    !Tr_meulage_bavure : Meulage de la bavure
    LOCAL CONST Robtarget Tr_meulage_bavure_0 := [[-72.96559375,77.9778671875,80.7656328125],[0.524498637144303,-0.433871580767109,0.466936666004684,-0.564470354382628],[0,0,0,0],[8.999999E+09,8.999999E+09,8.999999E+09,8.999999E+09,8.999999E+09,8.999999E+09]];
    LOCAL CONST Robtarget Tr_meulage_bavure_1 := [[-73.4128125,91.0669140625,78.9180078125],[0.519154027655531,-0.429298696043106,0.470963403699329,-0.569539460898604],[0,0,0,0],[8.999999E+09,8.999999E+09,8.999999E+09,8.999999E+09,8.999999E+09,8.999999E+09]];
    LOCAL CONST Robtarget Tr_meulage_bavure_2 := [[-73.421484375,92.5101640625,78.714984375],[0.502366205049294,-0.414981939275173,0.483103622109588,-0.584832519961385],[0,0,0,0],[8.999999E+09,8.999999E+09,8.999999E+09,8.999999E+09,8.999999E+09,8.999999E+09]];
    LOCAL CONST Robtarget Tr_meulage_bavure_3 := [[-73.3546796875,94.05434375,78.4991015625],[0.471901589556323,-0.389165581198061,0.503332600241078,-0.610340342529925],[0,0,0,0],[8.999999E+09,8.999999E+09,8.999999E+09,8.999999E+09,8.999999E+09,8.999999E+09]];
    LOCAL CONST Robtarget Tr_meulage_bavure_4 := [[-73.06753125,95.5965546875,78.2873359375],[0.424855473704573,-0.349592797660536,0.530576857987408,-0.644802993212153],[0,0,0,0],[8.999999E+09,8.999999E+09,8.999999E+09,8.999999E+09,8.999999E+09,8.999999E+09]];
    LOCAL CONST Robtarget Tr_meulage_bavure_5 := [[-72.49625,97.5792109375,78.0186171875],[0.360143668564367,-0.295563225119298,0.561336594654554,-0.683988410319727],[0,0,0,0],[8.999999E+09,8.999999E+09,8.999999E+09,8.999999E+09,8.999999E+09,8.999999E+09]];
    LOCAL CONST Robtarget Tr_meulage_bavure_6 := [[-71.18978125,99.7963125,77.72978125],[0.282652351555885,-0.231289577368078,0.589537581877902,-0.720456951603897],[0,0,0,0],[8.999999E+09,8.999999E+09,8.999999E+09,8.999999E+09,8.999999E+09,8.999999E+09]];
    LOCAL CONST Robtarget Tr_meulage_bavure_7 := [[-69.0200625,100.7901796875,77.627953125],[0.204414557432899,-0.166757138111491,0.609729609191989,-0.747419928335445],[0,0,0,0],[8.999999E+09,8.999999E+09,8.999999E+09,8.999999E+09,8.999999E+09,8.999999E+09]];
    LOCAL CONST Robtarget Tr_meulage_bavure_8 := [[-65.746828125,102.36953125,77.46309375],[0.137940363092354,-0.112187700081668,0.620915411831161,-0.763446414315291],[0,0,0,0],[8.999999E+09,8.999999E+09,8.999999E+09,8.999999E+09,8.999999E+09,8.999999E+09]];
    LOCAL CONST Robtarget Tr_meulage_bavure_9 := [[-61.93778515625,102.33946875,77.5338046875],[0.0895913508579802,-0.0726567540841667,0.625676522996422,-0.771507144820126],[0,0,0,0],[8.999999E+09,8.999999E+09,8.999999E+09,8.999999E+09,8.999999E+09,8.999999E+09]];
    LOCAL CONST Robtarget Tr_meulage_bavure_10 := [[-57.10214453125,102.293921875,77.6246171875],[0.0599889984484553,-0.0485258607399388,0.627036256816005,-0.775159398796642],[0,0,0,0],[8.999999E+09,8.999999E+09,8.999999E+09,8.999999E+09,8.999999E+09,8.999999E+09]];
    LOCAL CONST Robtarget Tr_meulage_bavure_11 := [[-55.68121484375,102.1337578125,77.6719296875],[0.047095653965774,-0.0380159924114396,0.626957544520652,-0.776698796875046],[0,0,0,0],[8.999999E+09,8.999999E+09,8.999999E+09,8.999999E+09,8.999999E+09,8.999999E+09]];
    LOCAL CONST Robtarget Tr_meulage_bavure_12 := [[-51.0949140625,101.74665625,77.8063984375],[0.0480334258632763,-0.0387120379923225,0.626315605146604,-0.777124784615805],[0,0,0,0],[8.999999E+09,8.999999E+09,8.999999E+09,8.999999E+09,8.999999E+09,8.999999E+09]];
    LOCAL CONST Robtarget Tr_meulage_bavure_13 := [[-49.12283984375,101.942609375,77.8132734375],[0.0593251793460015,-0.0477669656022839,0.625326539875387,-0.77663734047507],[0,0,0,0],[8.999999E+09,8.999999E+09,8.999999E+09,8.999999E+09,8.999999E+09,8.999999E+09]];
    LOCAL CONST Robtarget Tr_meulage_bavure_14 := [[-44.2636640625,102.2745859375,77.8514296875],[0.0768851540962994,-0.0618884366060826,0.62398012963373,-0.7751821026806],[0,0,0,0],[8.999999E+09,8.999999E+09,8.999999E+09,8.999999E+09,8.999999E+09,8.999999E+09]];
    LOCAL CONST Robtarget Tr_meulage_bavure_15 := [[-42.5008984375,102.301234375,77.878453125],[0.0961771542647169,-0.0774482725613951,0.622392974176696,-0.772902778989882],[0,0,0,0],[8.999999E+09,8.999999E+09,8.999999E+09,8.999999E+09,8.999999E+09,8.999999E+09]];
    LOCAL CONST Robtarget Tr_meulage_bavure_16 := [[-41.74234765625,102.4241171875,77.874421875],[0.112993286570119,-0.0910887399273819,0.620961489830233,-0.770287080766867],[0,0,0,0],[8.999999E+09,8.999999E+09,8.999999E+09,8.999999E+09,8.999999E+09,8.999999E+09]];
    LOCAL CONST Robtarget Tr_meulage_bavure_17 := [[-41.52457421875,102.525171875,77.864015625],[0.12430618580482,-0.100382813703911,0.620196366080517,-0.768002428631619],[0,0,0,0],[8.999999E+09,8.999999E+09,8.999999E+09,8.999999E+09,8.999999E+09,8.999999E+09]];
    LOCAL CONST Robtarget Tr_meulage_bavure_18 := [[-38.44026171875,103.5358046875,77.775796875],[0.128536780570744,-0.104042680848259,0.620496098458886,-0.766575507304868],[0,0,0,0],[8.999999E+09,8.999999E+09,8.999999E+09,8.999999E+09,8.999999E+09,8.999999E+09]];
    LOCAL CONST Robtarget Tr_meulage_bavure_19 := [[-35.635421875,105.1262265625,77.601203125],[0.125456426611608,-0.101841270384386,0.621966700070119,-0.766189574891376],[0,0,0,0],[8.999999E+09,8.999999E+09,8.999999E+09,8.999999E+09,8.999999E+09,8.999999E+09]];
    LOCAL CONST Robtarget Tr_meulage_bavure_20 := [[-32.589919921875,106.671859375,77.4371015625],[0.115819970243643,-0.0943317978781946,0.624426753397045,-0.766667122057451],[0,0,0,0],[8.999999E+09,8.999999E+09,8.999999E+09,8.999999E+09,8.999999E+09,8.999999E+09]];
    LOCAL CONST Robtarget Tr_meulage_bavure_21 := [[-30.991841796875,107.5399765625,77.3429765625],[0.1010430938105,-0.0826008420732401,0.627499640971008,-0.767601195063719],[0,0,0,0],[8.999999E+09,8.999999E+09,8.999999E+09,8.999999E+09,8.999999E+09,8.999999E+09]];
    LOCAL CONST Robtarget Tr_meulage_bavure_22 := [[-30.700533203125,107.67775,77.3286953125],[0.0830195632788944,-0.0681360313903383,0.630743998534626,-0.768522765864427],[0,0,0,0],[8.999999E+09,8.999999E+09,8.999999E+09,8.999999E+09,8.999999E+09,8.999999E+09]];
    LOCAL CONST Robtarget Tr_meulage_bavure_23 := [[-26.497271484375,109.0772421875,77.20534375],[0.0639091173605292,-0.0526684914647995,0.633792076669562,-0.769057382953902],[0,0,0,0],[8.999999E+09,8.999999E+09,8.999999E+09,8.999999E+09,8.999999E+09,8.999999E+09]];
    LOCAL CONST Robtarget Tr_meulage_bavure_24 := [[-26.031384765625,109.2446875,77.1899453125],[0.0458469341804628,-0.0379425139443275,0.63643994137898,-0.769027064074703],[0,0,0,0],[8.999999E+09,8.999999E+09,8.999999E+09,8.999999E+09,8.999999E+09,8.999999E+09]];
    LOCAL CONST Robtarget Tr_meulage_bavure_25 := [[-24.007275390625,109.3088125,77.2162578125],[0.0305658967448666,-0.0254025527691808,0.638653823464502,-0.768467130099371],[0,0,0,0],[8.999999E+09,8.999999E+09,8.999999E+09,8.999999E+09,8.999999E+09,8.999999E+09]];
    LOCAL CONST Robtarget Tr_meulage_bavure_26 := [[-22.2173125,109.3889609375,77.236234375],[0.0190622543195306,-0.015907517289484,0.640516947745874,-0.767542585791988],[0,0,0,0],[8.999999E+09,8.999999E+09,8.999999E+09,8.999999E+09,8.999999E+09,8.999999E+09]];
    LOCAL CONST Robtarget Tr_meulage_bavure_27 := [[-19.49805859375,109.3278828125,77.2922890625],[0.0115387164285388,-0.00966712028603791,0.642129419226901,-0.76644844169186],[0,0,0,0],[8.999999E+09,8.999999E+09,8.999999E+09,8.999999E+09,8.999999E+09,8.999999E+09]];
    LOCAL CONST Robtarget Tr_meulage_bavure_28 := [[-15.033275390625,109.3440546875,77.3679453125],[0.00752164158955457,-0.00632501640817029,0.643568832555467,-0.765325144522528],[0,0,0,0],[8.999999E+09,8.999999E+09,8.999999E+09,8.999999E+09,8.999999E+09,8.999999E+09]];
    LOCAL CONST Robtarget Tr_meulage_bavure_29 := [[-11.9529951171875,109.418640625,77.4112265625],[0.006151571426882,-0.00519059536474067,0.644865070540276,-0.764254052449723],[0,0,0,0],[8.999999E+09,8.999999E+09,8.999999E+09,8.999999E+09,8.999999E+09,8.999999E+09]];
    LOCAL CONST Robtarget Tr_meulage_bavure_30 := [[-3.52283715820313,109.6361953125,77.527796875],[0.00643709893464829,-0.00544820591259924,0.646018072081297,-0.763275527810242],[0,0,0,0],[8.999999E+09,8.999999E+09,8.999999E+09,8.999999E+09,8.999999E+09,8.999999E+09]];
    LOCAL CONST Robtarget Tr_meulage_bavure_31 := [[2.07959692382813,109.6801015625,77.619421875],[0.00754756157762624,-0.0064053255495668,0.647024086186714,-0.762405297734141],[0,0,0,0],[8.999999E+09,8.999999E+09,8.999999E+09,8.999999E+09,8.999999E+09,8.999999E+09]];
    LOCAL CONST Robtarget Tr_meulage_bavure_32 := [[10.4173935546875,109.9232578125,77.7307734375],[0.0089059924357084,-0.00757553932592323,0.64787449029423,-0.761657363470378],[0,0,0,0],[8.999999E+09,8.999999E+09,8.999999E+09,8.999999E+09,8.999999E+09,8.999999E+09]];
    LOCAL CONST Robtarget Tr_meulage_bavure_33 := [[14.9681103515625,110.080015625,77.788171875],[0.0101637625195787,-0.00866164743259205,0.648566021431958,-0.761041253572446],[0,0,0,0],[8.999999E+09,8.999999E+09,8.999999E+09,8.999999E+09,8.999999E+09,8.999999E+09]];
    LOCAL CONST Robtarget Tr_meulage_bavure_34 := [[17.49816015625,110.1214765625,77.8265078125],[0.011196506180603,-0.00955583886393558,0.649107385814113,-0.760554354319612],[0,0,0,0],[8.999999E+09,8.999999E+09,8.999999E+09,8.999999E+09,8.999999E+09,8.999999E+09]];
    LOCAL CONST Robtarget Tr_meulage_bavure_35 := [[19.417255859375,110.1771171875,77.8521875],[0.0119919328824449,-0.0102458555270846,0.649505699878697,-0.760193108239838],[0,0,0,0],[8.999999E+09,8.999999E+09,8.999999E+09,8.999999E+09,8.999999E+09,8.999999E+09]];
    LOCAL CONST Robtarget Tr_meulage_bavure_36 := [[28.539337890625,110.462484375,77.9713046875],[0.0126142416671802,-0.0107855693015085,0.64977613721374,-0.759944421592524],[0,0,0,0],[8.999999E+09,8.999999E+09,8.999999E+09,8.999999E+09,8.999999E+09,8.999999E+09]];
    LOCAL CONST Robtarget Tr_meulage_bavure_37 := [[30.24216796875,110.5603125,77.9872734375],[0.0132183794150829,-0.0113071132675388,0.64993291030976,-0.759792495179756],[0,0,0,0],[8.999999E+09,8.999999E+09,8.999999E+09,8.999999E+09,8.999999E+09,8.999999E+09]];
    LOCAL CONST Robtarget Tr_meulage_bavure_38 := [[35.8308828125,110.707703125,78.064109375],[0.0140329277622215,-0.0120062947243841,0.649995732976522,-0.759713415004451],[0,0,0,0],[8.999999E+09,8.999999E+09,8.999999E+09,8.999999E+09,8.999999E+09,8.999999E+09]];
    LOCAL CONST Robtarget Tr_meulage_bavure_39 := [[41.86768359375,110.7581015625,78.1623984375],[0.0153254201090454,-0.0131126639284937,0.649989769318002,-0.759675252542236],[0,0,0,0],[8.999999E+09,8.999999E+09,8.999999E+09,8.999999E+09,8.999999E+09,8.999999E+09]];
    LOCAL CONST Robtarget Tr_meulage_bavure_40 := [[48.0332890625,110.8994453125,78.2501484375],[0.0173576592937217,-0.0148509775353596,0.649939701863269,-0.759642379065289],[0,0,0,0],[8.999999E+09,8.999999E+09,8.999999E+09,8.999999E+09,8.999999E+09,8.999999E+09]];
    LOCAL CONST Robtarget Tr_meulage_bavure_41 := [[54.3366640625,111.20328125,78.31746875],[0.0203296694220353,-0.0173934789408263,0.649869936126184,-0.759574379209091],[0,0,0,0],[8.999999E+09,8.999999E+09,8.999999E+09,8.999999E+09,8.999999E+09,8.999999E+09]];
    LOCAL CONST Robtarget Tr_meulage_bavure_42 := [[62.10978125,111.67840625,78.386359375],[0.0243160425327989,-0.0208061051968355,0.649805737683987,-0.75942632251921],[0,0,0,0],[8.999999E+09,8.999999E+09,8.999999E+09,8.999999E+09,8.999999E+09,8.999999E+09]];
    LOCAL CONST Robtarget Tr_meulage_bavure_43 := [[64.7070625,111.7126171875,78.426890625],[0.0292129223072121,-0.0250039510309742,0.649775145993782,-0.759153256761685],[0,0,0,0],[8.999999E+09,8.999999E+09,8.999999E+09,8.999999E+09,8.999999E+09,8.999999E+09]];
    LOCAL CONST Robtarget Tr_meulage_bavure_44 := [[71.0410703125,111.980734375,78.499765625],[0.0346206886603777,-0.0296511906304267,0.649815638883284,-0.758723830041992],[0,0,0,0],[8.999999E+09,8.999999E+09,8.999999E+09,8.999999E+09,8.999999E+09,8.999999E+09]];
    LOCAL CONST Robtarget Tr_meulage_bavure_45 := [[73.262921875,112.0517265625,78.5285703125],[0.0397101679776423,-0.034045022612306,0.649985629173882,-0.758144261247124],[0,0,0,0],[8.999999E+09,8.999999E+09,8.999999E+09,8.999999E+09,8.999999E+09,8.999999E+09]];
    LOCAL CONST Robtarget Tr_meulage_bavure_46 := [[76.461375,112.383578125,78.53775],[0.0431961175728289,-0.037089230175035,0.6503823304321,-0.757470335190342],[0,0,0,0],[8.999999E+09,8.999999E+09,8.999999E+09,8.999999E+09,8.999999E+09,8.999999E+09]];
    LOCAL CONST Robtarget Tr_meulage_bavure_47 := [[79.9172578125,112.976390625,78.51475],[0.0432055408652098,-0.0371729766684629,0.651142540142572,-0.756812290770195],[0,0,0,0],[8.999999E+09,8.999999E+09,8.999999E+09,8.999999E+09,8.999999E+09,8.999999E+09]];
    LOCAL CONST Robtarget Tr_meulage_bavure_48 := [[80.2113828125,113.0060625,78.5157109375],[0.037391914390404,-0.0322554155127835,0.652386719553825,-0.756275744063048],[0,0,0,0],[8.999999E+09,8.999999E+09,8.999999E+09,8.999999E+09,8.999999E+09,8.999999E+09]];
    LOCAL CONST Robtarget Tr_meulage_bavure_49 := [[80.3745,113.014796875,78.517328125],[0.0230149202058911,-0.0199173517811249,0.654084723143131,-0.755808697685278],[0,0,0,0],[8.999999E+09,8.999999E+09,8.999999E+09,8.999999E+09,8.999999E+09,8.999999E+09]];
    LOCAL CONST Robtarget Tr_meulage_bavure_50 := [[80.4332421875,113.017515625,78.51796875],[0.00296501442514855,-0.00257573271942405,-0.655805220899747,0.754919920608174],[0,0,0,0],[8.999999E+09,8.999999E+09,8.999999E+09,8.999999E+09,8.999999E+09,8.999999E+09]];
    LOCAL CONST Robtarget Tr_meulage_bavure_51 := [[80.6750703125,113.011046875,78.5231015625],[0.0435007280531674,-0.0379546708906836,-0.656343344232936,0.752250320104651],[0,0,0,0],[8.999999E+09,8.999999E+09,8.999999E+09,8.999999E+09,8.999999E+09,8.999999E+09]];
    LOCAL CONST Robtarget Tr_meulage_bavure_52 := [[84.2401953125,113.0950625,78.5735234375],[0.100430419351731,-0.0880538690704243,-0.653348955544318,0.745181447232627],[0,0,0,0],[8.999999E+09,8.999999E+09,8.999999E+09,8.999999E+09,8.999999E+09,8.999999E+09]];
    LOCAL CONST Robtarget Tr_meulage_bavure_53 := [[87.07825,112.6916484375,78.679765625],[0.171895999689374,-0.151514363982637,-0.64363944210562,0.730221494728616],[0,0,0,0],[8.999999E+09,8.999999E+09,8.999999E+09,8.999999E+09,8.999999E+09,8.999999E+09]];
    LOCAL CONST Robtarget Tr_meulage_bavure_54 := [[87.4928984375,112.534953125,78.70903125],[0.249895133589002,-0.221511120301779,-0.625251119447997,0.70536960766694],[0,0,0,0],[8.999999E+09,8.999999E+09,8.999999E+09,8.999999E+09,8.999999E+09,8.999999E+09]];
    LOCAL CONST Robtarget Tr_meulage_bavure_55 := [[90.6231484375,111.0967890625,78.9658203125],[0.322554687399856,-0.287599923412569,-0.600154409759069,0.673096903971641],[0,0,0,0],[8.999999E+09,8.999999E+09,8.999999E+09,8.999999E+09,8.999999E+09,8.999999E+09]];
    LOCAL CONST Robtarget Tr_meulage_bavure_56 := [[91.76803125,109.5467734375,79.2036796875],[0.381349520380913,-0.342059463322267,-0.573448074256001,0.639316176073321],[0,0,0,0],[8.999999E+09,8.999999E+09,8.999999E+09,8.999999E+09,8.999999E+09,8.999999E+09]];
    LOCAL CONST Robtarget Tr_meulage_bavure_57 := [[92.15846875,108.9862109375,79.2892890625],[0.424645892808707,-0.383169856962373,-0.549520170935442,0.609002716062263],[0,0,0,0],[8.999999E+09,8.999999E+09,8.999999E+09,8.999999E+09,8.999999E+09,8.999999E+09]];
    LOCAL CONST Robtarget Tr_meulage_bavure_58 := [[92.243578125,108.7665078125,79.32165625],[0.455045695708042,-0.412995099011091,-0.530193694826248,0.584177292418059],[0,0,0,0],[8.999999E+09,8.999999E+09,8.999999E+09,8.999999E+09,8.999999E+09,8.999999E+09]];
    LOCAL CONST Robtarget Tr_meulage_bavure_59 := [[92.5548515625,106.992625,79.5764296875],[0.475960918078303,-0.43438038951089,-0.515492981292442,0.564837912952607],[0,0,0,0],[8.999999E+09,8.999999E+09,8.999999E+09,8.999999E+09,8.999999E+09,8.999999E+09]];
    LOCAL CONST Robtarget Tr_meulage_bavure_60 := [[93.0728125,104.701171875,79.9075625],[0.490145484495864,-0.449643756910361,-0.504780923350693,0.550249139318793],[0,0,0,0],[8.999999E+09,8.999999E+09,8.999999E+09,8.999999E+09,8.999999E+09,8.999999E+09]];
    LOCAL CONST Robtarget Tr_meulage_bavure_61 := [[93.1247578125,104.1366484375,79.9878203125],[0.499440463656121,-0.460329556127368,-0.497407243630099,0.539668376878659],[0,0,0,0],[8.999999E+09,8.999999E+09,8.999999E+09,8.999999E+09,8.999999E+09,8.999999E+09]];
    LOCAL CONST Robtarget Tr_meulage_bavure_62 := [[93.0234140625,101.6530390625,80.3351484375],[0.50508155139008,-0.467466020070269,-0.492804195180393,0.532458610351694],[0,0,0,0],[8.999999E+09,8.999999E+09,8.999999E+09,8.999999E+09,8.999999E+09,8.999999E+09]];
    LOCAL CONST Robtarget Tr_meulage_bavure_63 := [[93.0410859375,95.376796875,81.2176640625],[0.50800153503494,-0.471840804312682,-0.49042003163118,0.528004629110937],[0,0,0,0],[8.999999E+09,8.999999E+09,8.999999E+09,8.999999E+09,8.999999E+09,8.999999E+09]];
    LOCAL CONST Robtarget Tr_meulage_bavure_64 := [[93.069375,92.16809375,81.6691796875],[0.509036100077303,-0.474181488278619,-0.489639528685966,0.525630380533839],[0,0,0,0],[8.999999E+09,8.999999E+09,8.999999E+09,8.999999E+09,8.999999E+09,8.999999E+09]];
    LOCAL CONST Robtarget Tr_meulage_bavure_65 := [[93.288359375,82.485171875,83.0340546875],[0.509017334222879,-0.475239181311407,-0.489764889439004,0.524575473197039],[0,0,0,0],[8.999999E+09,8.999999E+09,8.999999E+09,8.999999E+09,8.999999E+09,8.999999E+09]];
    LOCAL CONST Robtarget Tr_meulage_bavure_66 := [[93.3151640625,82.0066953125,83.1017734375],[0.50860623912965,-0.475631289271055,-0.49021362642387,0.524199552320589],[0,0,0,0],[8.999999E+09,8.999999E+09,8.999999E+09,8.999999E+09,8.999999E+09,8.999999E+09]];
    LOCAL CONST Robtarget Tr_meulage_bavure_67 := [[93.3164765625,78.2097265625,83.6355078125],[0.508254924988694,-0.475792756551136,-0.490579965834165,0.524051029156855],[0,0,0,0],[8.999999E+09,8.999999E+09,8.999999E+09,8.999999E+09,8.999999E+09,8.999999E+09]];
    LOCAL CONST Robtarget Tr_meulage_bavure_68 := [[93.3254765625,77.7136796875,83.705390625],[0.508152417130769,-0.475929318394814,-0.490695448122873,0.523918297111197],[0,0,0,0],[8.999999E+09,8.999999E+09,8.999999E+09,8.999999E+09,8.999999E+09,8.999999E+09]];
    LOCAL CONST Robtarget Tr_meulage_bavure_69 := [[93.335359375,76.9299453125,83.8157265625],[0.508272125765174,-0.47604503540112,-0.490587023385963,0.523798570946311],[0,0,0,0],[8.999999E+09,8.999999E+09,8.999999E+09,8.999999E+09,8.999999E+09,8.999999E+09]];
    LOCAL CONST Robtarget Tr_meulage_bavure_70 := [[93.519703125,69.4331171875,84.87271875],[0.508492654218718,-0.476062116804073,-0.490368503184077,0.523773627280561],[0,0,0,0],[8.999999E+09,8.999999E+09,8.999999E+09,8.999999E+09,8.999999E+09,8.999999E+09]];
    LOCAL CONST Robtarget Tr_meulage_bavure_71 := [[93.6854296875,57.159515625,86.6008125],[0.508666271307918,-0.47588743567968,-0.490178457605301,0.523941650086731],[0,0,0,0],[8.999999E+09,8.999999E+09,8.999999E+09,8.999999E+09,8.999999E+09,8.999999E+09]];
    LOCAL CONST Robtarget Tr_meulage_bavure_72 := [[93.70446875,56.32636328125,86.7182578125],[0.508704393662726,-0.475482573374445,-0.490101155326875,0.524344371413212],[0,0,0,0],[8.999999E+09,8.999999E+09,8.999999E+09,8.999999E+09,8.999999E+09,8.999999E+09]];
    LOCAL CONST Robtarget Tr_meulage_bavure_73 := [[93.7035234375,55.86555859375,86.783015625],[0.508602047574567,-0.4748831497868,-0.490143997412789,0.524946485893312],[0,0,0,0],[8.999999E+09,8.999999E+09,8.999999E+09,8.999999E+09,8.999999E+09,8.999999E+09]];
    LOCAL CONST Robtarget Tr_meulage_bavure_74 := [[93.8570078125,51.93498046875,87.3381796875],[0.508420795232722,-0.474188979834551,-0.490254414881032,0.525645997861728],[0,0,0,0],[8.999999E+09,8.999999E+09,8.999999E+09,8.999999E+09,8.999999E+09,8.999999E+09]];
    LOCAL CONST Robtarget Tr_meulage_bavure_75 := [[94.0242734375,48.27883203125,87.855015625],[0.508263944010555,-0.473534553785341,-0.490342733317366,0.526304848422478],[0,0,0,0],[8.999999E+09,8.999999E+09,8.999999E+09,8.999999E+09,8.999999E+09,8.999999E+09]];
    LOCAL CONST Robtarget Tr_meulage_bavure_76 := [[94.0660078125,47.71273828125,87.9353203125],[0.50823520319336,-0.473057952864069,-0.49032064057548,0.526781568482337],[0,0,0,0],[8.999999E+09,8.999999E+09,8.999999E+09,8.999999E+09,8.999999E+09,8.999999E+09]];
    LOCAL CONST Robtarget Tr_meulage_bavure_77 := [[94.2361953125,44.8235,88.34440625],[0.508411095050095,-0.472850003528543,-0.490122652940176,0.526982748928183],[0,0,0,0],[8.999999E+09,8.999999E+09,8.999999E+09,8.999999E+09,8.999999E+09,8.999999E+09]];
    LOCAL CONST Robtarget Tr_meulage_bavure_78 := [[94.49140625,41.3637890625,88.8351640625],[0.508810216422261,-0.472937041493102,-0.489733748977065,0.526880986144834],[0,0,0,0],[8.999999E+09,8.999999E+09,8.999999E+09,8.999999E+09,8.999999E+09,8.999999E+09]];
    LOCAL CONST Robtarget Tr_meulage_bavure_79 := [[94.6926953125,36.78283203125,89.48259375],[0.509381048540969,-0.473309593721713,-0.489204041258047,0.526486829745137],[0,0,0,0],[8.999999E+09,8.999999E+09,8.999999E+09,8.999999E+09,8.999999E+09,8.999999E+09]];
    LOCAL CONST Robtarget Tr_meulage_bavure_80 := [[94.8668203125,33.4447890625,89.9548359375],[0.510042446720635,-0.473918883796655,-0.488608150999424,0.52585137529637],[0,0,0,0],[8.999999E+09,8.999999E+09,8.999999E+09,8.999999E+09,8.999999E+09,8.999999E+09]];
    LOCAL CONST Robtarget Tr_meulage_bavure_81 := [[94.8981484375,32.510306640625,90.086734375],[0.510736445760453,-0.474687805273883,-0.487994394189786,0.525053560825549],[0,0,0,0],[8.999999E+09,8.999999E+09,8.999999E+09,8.999999E+09,8.999999E+09,8.999999E+09]];
    LOCAL CONST Robtarget Tr_meulage_bavure_82 := [[94.9301796875,31.5094296875,90.2279765625],[0.511418105149978,-0.475576821233034,-0.487402262529341,0.524134756824968],[0,0,0,0],[8.999999E+09,8.999999E+09,8.999999E+09,8.999999E+09,8.999999E+09,8.999999E+09]];
    LOCAL CONST Robtarget Tr_meulage_bavure_83 := [[95.089,26.969724609375,90.868859375],[0.512034835099817,-0.476551606920003,-0.486879711480247,0.523131952890642],[0,0,0,0],[8.999999E+09,8.999999E+09,8.999999E+09,8.999999E+09,8.999999E+09,8.999999E+09]];
    LOCAL CONST Robtarget Tr_meulage_bavure_84 := [[95.22965625,22.79940625,91.4575078125],[0.512531744280155,-0.477540328865931,-0.486474082969998,0.522120112627602],[0,0,0,0],[8.999999E+09,8.999999E+09,8.999999E+09,8.999999E+09,8.999999E+09,8.999999E+09]];
    LOCAL CONST Robtarget Tr_meulage_bavure_85 := [[95.226046875,21.20137109375,91.6820625],[0.512784273545874,-0.478416827329453,-0.486298720705039,0.521232368884256],[0,0,0,0],[8.999999E+09,8.999999E+09,8.999999E+09,8.999999E+09,8.999999E+09,8.999999E+09]];
    LOCAL CONST Robtarget Tr_meulage_bavure_86 := [[95.44084375,11.85746875,92.9992109375],[0.51257251354118,-0.478964295880842,-0.486556288285653,0.520697224846776],[0,0,0,0],[8.999999E+09,8.999999E+09,8.999999E+09,8.999999E+09,8.999999E+09,8.999999E+09]];
    LOCAL CONST Robtarget Tr_meulage_bavure_87 := [[95.469671875,10.48285546875,93.1929375],[0.511662399007063,-0.478929085081936,-0.48746155010288,0.52077803148387],[0,0,0,0],[8.999999E+09,8.999999E+09,8.999999E+09,8.999999E+09,8.999999E+09,8.999999E+09]];
    LOCAL CONST Robtarget Tr_meulage_bavure_88 := [[95.47084375,9.393583984375,93.3460703125],[0.509916820225339,-0.478143213743958,-0.48913670941151,0.521640856440482],[0,0,0,0],[8.999999E+09,8.999999E+09,8.999999E+09,8.999999E+09,8.999999E+09,8.999999E+09]];
    LOCAL CONST Robtarget Tr_meulage_bavure_89 := [[95.3448359375,1.53523583984375,94.448453125],[0.507436151071227,-0.476663148416683,-0.491479978081437,0.523209543751435],[0,0,0,0],[8.999999E+09,8.999999E+09,8.999999E+09,8.999999E+09,8.999999E+09,8.999999E+09]];
    LOCAL CONST Robtarget Tr_meulage_bavure_90 := [[95.3131484375,0.499334686279297,94.5935078125],[0.504595584799778,-0.474839403042044,-0.494140253855218,0.525105938491602],[0,0,0,0],[8.999999E+09,8.999999E+09,8.999999E+09,8.999999E+09,8.999999E+09,8.999999E+09]];
    LOCAL CONST Robtarget Tr_meulage_bavure_91 := [[95.4977890625,-8.9034375,95.91840625],[0.501992798343004,-0.473193513735585,-0.496569781409481,0.52679178159997],[0,0,0,0],[8.999999E+09,8.999999E+09,8.999999E+09,8.999999E+09,8.999999E+09,8.999999E+09]];
    LOCAL CONST Robtarget Tr_meulage_bavure_92 := [[95.58446875,-9.3557177734375,95.9834921875],[0.500229194956659,-0.472222354742487,-0.498226528901943,0.527775639919839],[0,0,0,0],[8.999999E+09,8.999999E+09,8.999999E+09,8.999999E+09,8.999999E+09,8.999999E+09]];
    LOCAL CONST Robtarget Tr_meulage_bavure_93 := [[95.6886484375,-12.312650390625,96.4009453125],[0.499610422055294,-0.472202384573772,-0.498842983492434,0.52779732094521],[0,0,0,0],[8.999999E+09,8.999999E+09,8.999999E+09,8.999999E+09,8.999999E+09,8.999999E+09]];
    LOCAL CONST Robtarget Tr_meulage_bavure_94 := [[95.8067265625,-15.0403916015625,96.786421875],[0.500063158167775,-0.473050405070706,-0.49848329135892,0.526948346938948],[0,0,0,0],[8.999999E+09,8.999999E+09,8.999999E+09,8.999999E+09,8.999999E+09,8.999999E+09]];
    LOCAL CONST Robtarget Tr_meulage_bavure_95 := [[95.8925234375,-16.596419921875,97.006640625],[0.501240565163084,-0.474399052413705,-0.497448126220619,0.525593756263871],[0,0,0,0],[8.999999E+09,8.999999E+09,8.999999E+09,8.999999E+09,8.999999E+09,8.999999E+09]];
    LOCAL CONST Robtarget Tr_meulage_bavure_96 := [[96.1465546875,-22.8259375,97.8867109375],[0.50270497884405,-0.475784938551787,-0.496122644466237,0.524193397650622],[0,0,0,0],[8.999999E+09,8.999999E+09,8.999999E+09,8.999999E+09,8.999999E+09,8.999999E+09]];
    LOCAL CONST Robtarget Tr_meulage_bavure_97 := [[96.2089140625,-26.7219765625,98.4354375],[0.504123070686211,-0.476860966018335,-0.494807534813532,0.523095643435997],[0,0,0,0],[8.999999E+09,8.999999E+09,8.999999E+09,8.999999E+09,8.999999E+09,8.999999E+09]];
    LOCAL CONST Robtarget Tr_meulage_bavure_98 := [[96.2761328125,-32.718224609375,99.279453125],[0.505358446517146,-0.477499660830549,-0.493631604921573,0.522431577398457],[0,0,0,0],[8.999999E+09,8.999999E+09,8.999999E+09,8.999999E+09,8.999999E+09,8.999999E+09]];
    LOCAL CONST Robtarget Tr_meulage_bavure_99 := [[96.32565625,-36.04073828125,99.7473359375],[0.506481259161197,-0.477738348450034,-0.492531418727566,0.522164347791893],[0,0,0,0],[8.999999E+09,8.999999E+09,8.999999E+09,8.999999E+09,8.999999E+09,8.999999E+09]];
    LOCAL CONST Robtarget Tr_meulage_bavure_100 := [[96.58703125,-43.539609375,100.8059609375],[0.507646887961661,-0.477718557261596,-0.491365597045757,0.522148893736841],[0,0,0,0],[8.999999E+09,8.999999E+09,8.999999E+09,8.999999E+09,8.999999E+09,8.999999E+09]];
    LOCAL CONST Robtarget Tr_meulage_bavure_101 := [[96.742390625,-46.9201328125,101.28384375],[0.508967667396993,-0.477569831764066,-0.490033634824307,0.522250903373257],[0,0,0,0],[8.999999E+09,8.999999E+09,8.999999E+09,8.999999E+09,8.999999E+09,8.999999E+09]];
    LOCAL CONST Robtarget Tr_meulage_bavure_102 := [[96.6823671875,-48.3631484375,101.4856328125],[0.510473405211254,-0.477337868130739,-0.488509837846581,0.522420903628038],[0,0,0,0],[8.999999E+09,8.999999E+09,8.999999E+09,8.999999E+09,8.999999E+09,8.999999E+09]];
    LOCAL CONST Robtarget Tr_meulage_bavure_103 := [[96.7233359375,-51.52609375,101.9309375],[0.512066075876696,-0.476986193405036,-0.486888647820034,0.522696804908155],[0,0,0,0],[8.999999E+09,8.999999E+09,8.999999E+09,8.999999E+09,8.999999E+09,8.999999E+09]];
    LOCAL CONST Robtarget Tr_meulage_bavure_104 := [[96.7839921875,-58.093375,102.855109375],[0.513578282717062,-0.47639084711756,-0.485325101705186,0.523209952083156],[0,0,0,0],[8.999999E+09,8.999999E+09,8.999999E+09,8.999999E+09,8.999999E+09,8.999999E+09]];
    LOCAL CONST Robtarget Tr_meulage_bavure_105 := [[96.821171875,-61.7732578125,103.3730078125],[0.514764031038119,-0.47539080126442,-0.484047150576434,0.524137324030062],[0,0,0,0],[8.999999E+09,8.999999E+09,8.999999E+09,8.999999E+09,8.999999E+09,8.999999E+09]];
    LOCAL CONST Robtarget Tr_meulage_bavure_106 := [[96.848578125,-65.96228125,103.9623046875],[0.515341410888379,-0.47383806037692,-0.483315501544715,0.525648978623942],[0,0,0,0],[8.999999E+09,8.999999E+09,8.999999E+09,8.999999E+09,8.999999E+09,8.999999E+09]];
    LOCAL CONST Robtarget Tr_meulage_bavure_107 := [[96.9078515625,-71.838828125,104.789359375],[0.515050095490584,-0.471555521273802,-0.48335891084395,0.527942186985548],[0,0,0,0],[8.999999E+09,8.999999E+09,8.999999E+09,8.999999E+09,8.999999E+09,8.999999E+09]];
    LOCAL CONST Robtarget Tr_meulage_bavure_108 := [[97.005765625,-76.6273125,105.4641484375],[0.513578845853097,-0.468354543928388,-0.48444310717155,0.531220920322051],[0,0,0,0],[8.999999E+09,8.999999E+09,8.999999E+09,8.999999E+09,8.999999E+09,8.999999E+09]];
    LOCAL CONST Robtarget Tr_meulage_bavure_109 := [[97.0657421875,-80.4912578125,106.0083203125],[0.510678605778018,-0.464109782623466,-0.486762395276764,0.535604183906591],[0,0,0,0],[8.999999E+09,8.999999E+09,8.999999E+09,8.999999E+09,8.999999E+09,8.999999E+09]];
    LOCAL CONST Robtarget Tr_meulage_bavure_110 := [[97.18928125,-83.593078125,106.4464765625],[0.506351626893115,-0.458888369224079,-0.4902729646951,0.54098236073151],[0,0,0,0],[8.999999E+09,8.999999E+09,8.999999E+09,8.999999E+09,8.999999E+09,8.999999E+09]];
    LOCAL CONST Robtarget Tr_meulage_bavure_111 := [[97.30415625,-86.67925,106.88228125],[0.501083028037151,-0.453206449217312,-0.494530085943956,0.546772080027153],[0,0,0,0],[8.999999E+09,8.999999E+09,8.999999E+09,8.999999E+09,8.999999E+09,8.999999E+09]];
    LOCAL CONST Robtarget Tr_meulage_bavure_112 := [[97.352984375,-91.204046875,107.5191484375],[0.496010154722637,-0.448147678011833,-0.498598331813601,0.551848972652231],[0,0,0,0],[8.999999E+09,8.999999E+09,8.999999E+09,8.999999E+09,8.999999E+09,8.999999E+09]];
    LOCAL CONST Robtarget Tr_meulage_bavure_113 := [[97.4324140625,-95.1215234375,108.0711875],[0.49268192858625,-0.445141272111876,-0.501284971831372,0.554821721026831],[0,0,0,0],[8.999999E+09,8.999999E+09,8.999999E+09,8.999999E+09,8.999999E+09,8.999999E+09]];
    LOCAL CONST Robtarget Tr_meulage_bavure_114 := [[97.4640234375,-95.146828125,108.0752890625],[0.492284416657108,-0.445263315632892,-0.501710204049278,0.554692260646394],[0,0,0,0],[8.999999E+09,8.999999E+09,8.999999E+09,8.999999E+09,8.999999E+09,8.999999E+09]];
    LOCAL CONST Robtarget Tr_meulage_bavure_115 := [[97.6526953125,-102.9675859375,109.177890625],[0.494768114057018,-0.448481249387066,-0.499910727661733,0.551505527288162],[0,0,0,0],[8.999999E+09,8.999999E+09,8.999999E+09,8.999999E+09,8.999999E+09,8.999999E+09]];
    LOCAL CONST Robtarget Tr_meulage_bavure_116 := [[97.7313984375,-107.320109375,109.7910625],[0.498868251909272,-0.453686160536239,-0.496832755859474,0.546311767839531],[0,0,0,0],[8.999999E+09,8.999999E+09,8.999999E+09,8.999999E+09,8.999999E+09,8.999999E+09]];
    LOCAL CONST Robtarget Tr_meulage_bavure_117 := [[97.7648203125,-111.517140625,110.38159375],[0.503018852075786,-0.459452841372573,-0.493691118633628,0.540503654375533],[0,0,0,0],[8.999999E+09,8.999999E+09,8.999999E+09,8.999999E+09,8.999999E+09,8.999999E+09]];
    LOCAL CONST Robtarget Tr_meulage_bavure_118 := [[97.8033046875,-112.682703125,110.54609375],[0.506131659737862,-0.464747121213921,-0.491387390034454,0.535144176133402],[0,0,0,0],[8.999999E+09,8.999999E+09,8.999999E+09,8.999999E+09,8.999999E+09,8.999999E+09]];
    LOCAL CONST Robtarget Tr_meulage_bavure_119 := [[97.84084375,-114.373328125,110.784390625],[0.507813569410199,-0.469157423878958,-0.490291564577917,0.530689054009852],[0,0,0,0],[8.999999E+09,8.999999E+09,8.999999E+09,8.999999E+09,8.999999E+09,8.999999E+09]];
    LOCAL CONST Robtarget Tr_meulage_bavure_120 := [[98.15975,-122.4149140625,111.920296875],[0.508195885932996,-0.472735439316485,-0.490325003028154,0.527104863704053],[0,0,0,0],[8.999999E+09,8.999999E+09,8.999999E+09,8.999999E+09,8.999999E+09,8.999999E+09]];
    LOCAL CONST Robtarget Tr_meulage_bavure_121 := [[98.3548203125,-126.0976796875,112.441359375],[0.507667580035712,-0.475761230067035,-0.491163294208522,0.524102564931731],[0,0,0,0],[8.999999E+09,8.999999E+09,8.999999E+09,8.999999E+09,8.999999E+09,8.999999E+09]];
    LOCAL CONST Robtarget Tr_meulage_bavure_122 := [[98.4237109375,-133.3633125,113.4638359375],[0.506682046015217,-0.478576480590122,-0.492403964431644,0.521321582407448],[0,0,0,0],[8.999999E+09,8.999999E+09,8.999999E+09,8.999999E+09,8.999999E+09,8.999999E+09]];
    LOCAL CONST Robtarget Tr_meulage_bavure_123 := [[98.6452109375,-145.5534375,115.1811796875],[0.50574841062659,-0.481609606428448,-0.493577670608932,0.518316327372362],[0,0,0,0],[8.999999E+09,8.999999E+09,8.999999E+09,8.999999E+09,8.999999E+09,8.999999E+09]];
    LOCAL CONST Robtarget Tr_meulage_bavure_124 := [[98.66753125,-147.15303125,115.40640625],[0.505558330250797,-0.485444325289496,-0.494019781185393,0.51448910343737],[0,0,0,0],[8.999999E+09,8.999999E+09,8.999999E+09,8.999999E+09,8.999999E+09,8.999999E+09]];
    LOCAL CONST Robtarget Tr_meulage_bavure_125 := [[98.701515625,-148.2614375,115.5628046875],[0.507039868917661,-0.490930875802081,-0.492797454411434,0.508967695868583],[0,0,0,0],[8.999999E+09,8.999999E+09,8.999999E+09,8.999999E+09,8.999999E+09,8.999999E+09]];
    LOCAL CONST Robtarget Tr_meulage_bavure_126 := [[98.9204765625,-152.394078125,116.147515625],[0.511327904645476,-0.499196706833558,-0.488671184252742,0.500546596730435],[0,0,0,0],[8.999999E+09,8.999999E+09,8.999999E+09,8.999999E+09,8.999999E+09,8.999999E+09]];
    LOCAL CONST Robtarget Tr_meulage_bavure_127 := [[99.1385703125,-155.905109375,116.64484375],[0.519577232756094,-0.51138843510594,-0.48014531891565,0.487833824539471],[0,0,0,0],[8.999999E+09,8.999999E+09,8.999999E+09,8.999999E+09,8.999999E+09,8.999999E+09]];
    LOCAL CONST Robtarget Tr_meulage_bavure_128 := [[99.268203125,-158.178890625,116.9667109375],[0.532651208428772,-0.528416135275659,-0.465601888439109,0.469333527058999],[0,0,0,0],[8.999999E+09,8.999999E+09,8.999999E+09,8.999999E+09,8.999999E+09,8.999999E+09]];
    LOCAL CONST Robtarget Tr_meulage_bavure_129 := [[98.884234375,-161.558140625,117.4350078125],[0.550786855280955,-0.550601613333312,-0.443474547099509,0.443623747695449],[0,0,0,0],[8.999999E+09,8.999999E+09,8.999999E+09,8.999999E+09,8.999999E+09,8.999999E+09]];
    LOCAL CONST Robtarget Tr_meulage_bavure_130 := [[98.8758984375,-161.623609375,117.4440625],[0.573338153790971,-0.577382144069585,-0.412485306911119,0.409596255719715],[0,0,0,0],[8.999999E+09,8.999999E+09,8.999999E+09,8.999999E+09,8.999999E+09,8.999999E+09]];
    LOCAL CONST Robtarget Tr_meulage_bavure_131 := [[97.341453125,-164.4365,117.8126640625],[0.598589585207786,-0.607108569462481,-0.372134968749448,0.366913148306022],[0,0,0,0],[8.999999E+09,8.999999E+09,8.999999E+09,8.999999E+09,8.999999E+09,8.999999E+09]];
    LOCAL CONST Robtarget Tr_meulage_bavure_132 := [[97.3365859375,-164.444078125,117.8136484375],[0.623860751882062,-0.637046977120005,-0.323462099081456,0.316766762241921],[0,0,0,0],[8.999999E+09,8.999999E+09,8.999999E+09,8.999999E+09,8.999999E+09,8.999999E+09]];
    LOCAL CONST Robtarget Tr_meulage_bavure_133 := [[97.3249765625,-164.45096875,117.8144140625],[0.646136841065887,-0.664081727399951,-0.269608961330264,0.26232355960018],[0,0,0,0],[8.999999E+09,8.999999E+09,8.999999E+09,8.999999E+09,8.999999E+09,8.999999E+09]];
    LOCAL CONST Robtarget Tr_meulage_bavure_134 := [[94.8720546875,-165.7548125,117.9548671875],[0.663195970054067,-0.685877063949421,-0.215360759525238,0.208239049433287],[0,0,0,0],[8.999999E+09,8.999999E+09,8.999999E+09,8.999999E+09,8.999999E+09,8.999999E+09]];
    LOCAL CONST Robtarget Tr_meulage_bavure_135 := [[94.5723359375,-165.84928125,117.9629140625],[0.674467278413093,-0.701723788105488,-0.165474224209869,0.159046838003974],[0,0,0,0],[8.999999E+09,8.999999E+09,8.999999E+09,8.999999E+09,8.999999E+09,8.999999E+09]];
    LOCAL CONST Robtarget Tr_meulage_bavure_136 := [[93.1553203125,-166.2681875,117.9970625],[0.680830218689629,-0.71240263778997,-0.123012663707437,0.117560961022465],[0,0,0,0],[8.999999E+09,8.999999E+09,8.999999E+09,8.999999E+09,8.999999E+09,8.999999E+09]];
    LOCAL CONST Robtarget Tr_meulage_bavure_137 := [[92.3421015625,-166.301921875,117.987609375],[0.683734509021044,-0.719328021473193,-0.0889905916596248,0.0845871934354406],[0,0,0,0],[8.999999E+09,8.999999E+09,8.999999E+09,8.999999E+09,8.999999E+09,8.999999E+09]];
    LOCAL CONST Robtarget Tr_meulage_bavure_138 := [[83.7809453125,-166.49628125,117.8654921875],[0.684477059249715,-0.723856009871078,-0.0630239878092534,0.0595953798125553],[0,0,0,0],[8.999999E+09,8.999999E+09,8.999999E+09,8.999999E+09,8.999999E+09,8.999999E+09]];
    LOCAL CONST Robtarget Tr_meulage_bavure_139 := [[82.838203125,-166.5025625,117.849921875],[0.684005504642971,-0.726965777387181,-0.0440438834567159,0.0414410962212351],[0,0,0,0],[8.999999E+09,8.999999E+09,8.999999E+09,8.999999E+09,8.999999E+09,8.999999E+09]];
    LOCAL CONST Robtarget Tr_meulage_bavure_140 := [[81.850546875,-166.521203125,117.835296875],[0.682945401717553,-0.729250006727333,-0.0307945624667288,0.028839224738492],[0,0,0,0],[8.999999E+09,8.999999E+09,8.999999E+09,8.999999E+09,8.999999E+09,8.999999E+09]];
    LOCAL CONST Robtarget Tr_meulage_bavure_141 := [[74.306140625,-166.74209375,117.7346640625],[0.681637040893357,-0.731072769865234,-0.0219853259932027,0.0204986605585721],[0,0,0,0],[8.999999E+09,8.999999E+09,8.999999E+09,8.999999E+09,8.999999E+09,8.999999E+09]];
    LOCAL CONST Robtarget Tr_meulage_bavure_142 := [[73.7237890625,-166.75646875,117.726515625],[0.680254493972394,-0.732632448263654,-0.0164438506926185,0.0152682335574622],[0,0,0,0],[8.999999E+09,8.999999E+09,8.999999E+09,8.999999E+09,8.999999E+09,8.999999E+09]];
    LOCAL CONST Robtarget Tr_meulage_bavure_143 := [[71.5945859375,-166.840625,117.7011796875],[0.678885847668454,-0.734026017031106,-0.0131289016534278,0.0121426561472485],[0,0,0,0],[8.999999E+09,8.999999E+09,8.999999E+09,8.999999E+09,8.999999E+09,8.999999E+09]];
    LOCAL CONST Robtarget Tr_meulage_bavure_144 := [[63.42403515625,-167.19125,117.60784375],[0.677571719896211,-0.735299717926155,-0.011174198072345,0.0102969175993891],[0,0,0,0],[8.999999E+09,8.999999E+09,8.999999E+09,8.999999E+09,8.999999E+09,8.999999E+09]];
    LOCAL CONST Robtarget Tr_meulage_bavure_145 := [[60.74982421875,-167.22803125,117.56634375],[0.676332886541328,-0.73647111859363,-0.00999410481574146,0.00917801335011573],[0,0,0,0],[8.999999E+09,8.999999E+09,8.999999E+09,8.999999E+09,8.999999E+09,8.999999E+09]];
    LOCAL CONST Robtarget Tr_meulage_bavure_146 := [[57.07700390625,-167.319140625,117.5150390625],[0.675163263386652,-0.737562914117785,-0.0091985563275435,0.00842033566177708],[0,0,0,0],[8.999999E+09,8.999999E+09,8.999999E+09,8.999999E+09,8.999999E+09,8.999999E+09]];
    LOCAL CONST Robtarget Tr_meulage_bavure_147 := [[54.9374921875,-167.37096875,117.4849765625],[0.674076549603267,-0.738570889782252,-0.00854523514019493,0.00779903824878532],[0,0,0,0],[8.999999E+09,8.999999E+09,8.999999E+09,8.999999E+09,8.999999E+09,8.999999E+09]];
    LOCAL CONST Robtarget Tr_meulage_bavure_148 := [[49.7376484375,-167.550609375,117.4194609375],[0.67307174839465,-0.739499761318672,-0.00791429352454091,0.00720336592181224],[0,0,0,0],[8.999999E+09,8.999999E+09,8.999999E+09,8.999999E+09,8.999999E+09,8.999999E+09]];
    LOCAL CONST Robtarget Tr_meulage_bavure_149 := [[47.34811328125,-167.626484375,117.388421875],[0.672108949669749,-0.740386315879231,-0.00731719610483644,0.00664241475439612],[0,0,0,0],[8.999999E+09,8.999999E+09,8.999999E+09,8.999999E+09,8.999999E+09,8.999999E+09]];
    LOCAL CONST Robtarget Tr_meulage_bavure_150 := [[35.66473828125,-167.939203125,117.2284453125],[0.671196190990874,-0.741221936327509,-0.00686267661317515,0.0062143363235948],[0,0,0,0],[8.999999E+09,8.999999E+09,8.999999E+09,8.999999E+09,8.999999E+09,8.999999E+09]];
    LOCAL CONST Robtarget Tr_meulage_bavure_151 := [[31.9954375,-168.01475,117.175015625],[0.670336338775432,-0.742002296101295,-0.00671059701720467,0.00606245702896884],[0,0,0,0],[8.999999E+09,8.999999E+09,8.999999E+09,8.999999E+09,8.999999E+09,8.999999E+09]];
    LOCAL CONST Robtarget Tr_meulage_bavure_152 := [[28.97093359375,-168.014578125,117.1221953125],[0.669500961278734,-0.742751539665752,-0.00699216941986249,0.00630259770330242],[0,0,0,0],[8.999999E+09,8.999999E+09,8.999999E+09,8.999999E+09,8.999999E+09,8.999999E+09]];
    LOCAL CONST Robtarget Tr_meulage_bavure_153 := [[28.38337109375,-168.02940625,117.1140234375],[0.66868380710914,-0.743474500117858,-0.00771371797956261,0.0069377474341386],[0,0,0,0],[8.999999E+09,8.999999E+09,8.999999E+09,8.999999E+09,8.999999E+09,8.999999E+09]];
    LOCAL CONST Robtarget Tr_meulage_bavure_154 := [[20.670576171875,-168.332546875,117.0220078125],[0.667875250109066,-0.744180886329373,-0.00872558392603669,0.00783089387809151],[0,0,0,0],[8.999999E+09,8.999999E+09,8.999999E+09,8.999999E+09,8.999999E+09,8.999999E+09]];
    LOCAL CONST Robtarget Tr_meulage_bavure_155 := [[19.9416171875,-168.335015625,117.0096328125],[0.667059330305528,-0.744888995955516,-0.00977660000248018,0.00875509275305352],[0,0,0,0],[8.999999E+09,8.999999E+09,8.999999E+09,8.999999E+09,8.999999E+09,8.999999E+09]];
    LOCAL CONST Robtarget Tr_meulage_bavure_156 := [[17.17451171875,-168.40121875,116.9706328125],[0.666263312393413,-0.745580824230547,-0.010609122230091,0.00948048647294788],[0,0,0,0],[8.999999E+09,8.999999E+09,8.999999E+09,8.999999E+09,8.999999E+09,8.999999E+09]];
    LOCAL CONST Robtarget Tr_meulage_bavure_157 := [[10.0085185546875,-168.699828125,116.8875234375],[0.665470091751805,-0.746277050711341,-0.0110733289179768,0.0098743076770483],[0,0,0,0],[8.999999E+09,8.999999E+09,8.999999E+09,8.999999E+09,8.999999E+09,8.999999E+09]];
    LOCAL CONST Robtarget Tr_meulage_bavure_158 := [[9.380119140625,-168.718703125,116.8792109375],[0.664674932797161,-0.746983105245555,-0.011167938053073,0.00993737130436034],[0,0,0,0],[8.999999E+09,8.999999E+09,8.999999E+09,8.999999E+09,8.999999E+09,8.999999E+09]];
    LOCAL CONST Robtarget Tr_meulage_bavure_159 := [[6.4452802734375,-168.836609375,116.8445546875],[0.663892088895315,-0.747682990160976,-0.0110264310833663,0.00979072743572814],[0,0,0,0],[8.999999E+09,8.999999E+09,8.999999E+09,8.999999E+09,8.999999E+09,8.999999E+09]];
    LOCAL CONST Robtarget Tr_meulage_bavure_160 := [[2.91008959960938,-168.9083125,116.7929296875],[0.66312720454389,-0.748366040344425,-0.0108609702726936,0.00962390657418241],[0,0,0,0],[8.999999E+09,8.999999E+09,8.999999E+09,8.999999E+09,8.999999E+09,8.999999E+09]];
    LOCAL CONST Robtarget Tr_meulage_bavure_161 := [[-4.9102626953125,-169.111546875,116.6849921875],[0.66237258499227,-0.749033736993813,-0.0108819943641858,0.00962297741862143],[0,0,0,0],[8.999999E+09,8.999999E+09,8.999999E+09,8.999999E+09,8.999999E+09,8.999999E+09]];
    LOCAL CONST Robtarget Tr_meulage_bavure_162 := [[-6.49701611328125,-169.132125,116.6601875],[0.661651542963285,-0.749662357417219,-0.0112107880615082,0.00989463475835567],[0,0,0,0],[8.999999E+09,8.999999E+09,8.999999E+09,8.999999E+09,8.999999E+09,8.999999E+09]];
    LOCAL CONST Robtarget Tr_meulage_bavure_163 := [[-9.96698828125,-169.223953125,116.6125234375],[0.660966621821724,-0.750249648423375,-0.0118304566539753,0.010422579984701],[0,0,0,0],[8.999999E+09,8.999999E+09,8.999999E+09,8.999999E+09,8.999999E+09,8.999999E+09]];
    LOCAL CONST Robtarget Tr_meulage_bavure_164 := [[-17.966248046875,-169.443765625,116.503796875],[0.660332626786627,-0.750787473448942,-0.0125421866810416,0.0110311044997792],[0,0,0,0],[8.999999E+09,8.999999E+09,8.999999E+09,8.999999E+09,8.999999E+09,8.999999E+09]];
    LOCAL CONST Robtarget Tr_meulage_bavure_165 := [[-20.5874921875,-169.518984375,116.468609375],[0.659752580805589,-0.751284870779714,-0.0129618661905187,0.0113826658886078],[0,0,0,0],[8.999999E+09,8.999999E+09,8.999999E+09,8.999999E+09,8.999999E+09,8.999999E+09]];
    LOCAL CONST Robtarget Tr_meulage_bavure_166 := [[-20.7209375,-169.524171875,116.467015625],[0.659250388328633,-0.751736307637985,-0.0126132415345911,0.0110614377611869],[0,0,0,0],[8.999999E+09,8.999999E+09,8.999999E+09,8.999999E+09,8.999999E+09,8.999999E+09]];
    LOCAL CONST Robtarget Tr_meulage_bavure_167 := [[-21.022080078125,-169.540546875,116.4640546875],[0.658854674864978,-0.752125322507375,-0.0111066322020573,0.00972930485033575],[0,0,0,0],[8.999999E+09,8.999999E+09,8.999999E+09,8.999999E+09,8.999999E+09,8.999999E+09]];
    LOCAL CONST Robtarget Tr_meulage_bavure_168 := [[-28.000173828125,-169.83925,116.3842421875],[0.658544361464871,-0.752460428129826,-0.00833307445557178,0.00729300703562969],[0,0,0,0],[8.999999E+09,8.999999E+09,8.999999E+09,8.999999E+09,8.999999E+09,8.999999E+09]];
    LOCAL CONST Robtarget Tr_meulage_bavure_169 := [[-29.79684375,-169.9663125,116.3707421875],[0.658298079979653,-0.752732618817936,-0.00459375700280629,0.0040174443610393],[0,0,0,0],[8.999999E+09,8.999999E+09,8.999999E+09,8.999999E+09,8.999999E+09,8.999999E+09]];
    LOCAL CONST Robtarget Tr_meulage_bavure_170 := [[-32.52297265625,-170.0338125,116.332640625],[0.658125935272267,-0.752907432831256,-0.000607438081315007,0.000530969330296183],[0,0,0,0],[8.999999E+09,8.999999E+09,8.999999E+09,8.999999E+09,8.999999E+09,8.999999E+09]];
    LOCAL CONST Robtarget Tr_meulage_bavure_171 := [[-32.742830078125,-170.038578125,116.3294765625],[0.658016379434283,-0.752995118377619,0.00269360356771767,-0.00235384695597986],[0,0,0,0],[8.999999E+09,8.999999E+09,8.999999E+09,8.999999E+09,8.999999E+09,8.999999E+09]];
    LOCAL CONST Robtarget Tr_meulage_bavure_172 := [[-32.91678125,-170.036515625,116.3261484375],[0.657980016469929,-0.753012170808398,0.00445295537875365,-0.00389098047420233],[0,0,0,0],[8.999999E+09,8.999999E+09,8.999999E+09,8.999999E+09,8.999999E+09,8.999999E+09]];
    LOCAL CONST Robtarget Tr_meulage_bavure_173 := [[-33.09648828125,-170.03040625,116.32215625],[0.658003378884216,-0.752994573902908,0.004173926680005,-0.00364738067689237],[0,0,0,0],[8.999999E+09,8.999999E+09,8.999999E+09,8.999999E+09,8.999999E+09,8.999999E+09]];
    LOCAL CONST Robtarget Tr_meulage_bavure_174 := [[-35.40748046875,-169.921078125,116.2664453125],[0.658098488449272,-0.752927855470324,0.00184797302504738,-0.00161522547697353],[0,0,0,0],[8.999999E+09,8.999999E+09,8.999999E+09,8.999999E+09,8.999999E+09,8.999999E+09]];
    LOCAL CONST Robtarget Tr_meulage_bavure_175 := [[-41.99823828125,-170.0676875,116.172015625],[0.658242652747245,-0.752800914933211,-0.00204682050810798,0.00178972226816966],[0,0,0,0],[8.999999E+09,8.999999E+09,8.999999E+09,8.999999E+09,8.999999E+09,8.999999E+09]];
    LOCAL CONST Robtarget Tr_meulage_bavure_176 := [[-44.52558984375,-170.152734375,116.1398515625],[0.658402823111578,-0.752613365370111,-0.00668306268505166,0.00584649109533925],[0,0,0,0],[8.999999E+09,8.999999E+09,8.999999E+09,8.999999E+09,8.999999E+09,8.999999E+09]];
    LOCAL CONST Robtarget Tr_meulage_bavure_177 := [[-45.7160703125,-170.18525,116.123640625],[0.658593449850906,-0.752354450158747,-0.0110955431006766,0.00971277834151459],[0,0,0,0],[8.999999E+09,8.999999E+09,8.999999E+09,8.999999E+09,8.999999E+09,8.999999E+09]];
    LOCAL CONST Robtarget Tr_meulage_bavure_178 := [[-50.14087890625,-170.324859375,116.06603125],[0.658832131354734,-0.75204605192743,-0.0144089586620694,0.0126230101489177],[0,0,0,0],[8.999999E+09,8.999999E+09,8.999999E+09,8.999999E+09,8.999999E+09,8.999999E+09]];
    LOCAL CONST Robtarget Tr_meulage_bavure_179 := [[-54.33327734375,-170.705109375,116.0463046875],[0.659149818217803,-0.751709467333879,-0.016027468863844,0.0140539711779391],[0,0,0,0],[8.999999E+09,8.999999E+09,8.999999E+09,8.999999E+09,8.999999E+09,8.999999E+09]];
    LOCAL CONST Robtarget Tr_meulage_bavure_180 := [[-54.73071484375,-170.743203125,116.04471875],[0.659590822483465,-0.751336056884888,-0.0156571119824787,0.0137452306136575],[0,0,0,0],[8.999999E+09,8.999999E+09,8.999999E+09,8.999999E+09,8.999999E+09,8.999999E+09]];
    LOCAL CONST Robtarget Tr_meulage_bavure_181 := [[-60.2934453125,-170.89784375,115.969359375],[0.660141420276806,-0.750931788056189,-0.0133246286033797,0.0117136328369653],[0,0,0,0],[8.999999E+09,8.999999E+09,8.999999E+09,8.999999E+09,8.999999E+09,8.999999E+09]];
    LOCAL CONST Robtarget Tr_meulage_bavure_182 := [[-62.477421875,-170.916265625,115.933828125],[0.660840818788693,-0.750426987692258,-0.00915307136530318,0.00806037532589221],[0,0,0,0],[8.999999E+09,8.999999E+09,8.999999E+09,8.999999E+09,8.999999E+09,8.999999E+09]];
    LOCAL CONST Robtarget Tr_meulage_bavure_183 := [[-65.7071484375,-170.87721875,115.8719609375],[0.661677235952261,-0.749778265783744,-0.00297916165751976,0.00262910188379773],[0,0,0,0],[8.999999E+09,8.999999E+09,8.999999E+09,8.999999E+09,8.999999E+09,8.999999E+09]];
    LOCAL CONST Robtarget Tr_meulage_bavure_184 := [[-68.5179765625,-170.8676875,115.8215625],[0.662617167733076,-0.748918083568882,0.00581059823691412,-0.00514101906610554],[0,0,0,0],[8.999999E+09,8.999999E+09,8.999999E+09,8.999999E+09,8.999999E+09,8.999999E+09]];
    LOCAL CONST Robtarget Tr_meulage_bavure_185 := [[-72.864546875,-170.853140625,115.7436484375],[0.663592641097019,-0.747682850338995,0.0185500800475915,-0.0164637942488065],[0,0,0,0],[8.999999E+09,8.999999E+09,8.999999E+09,8.999999E+09,8.999999E+09,8.999999E+09]];
    LOCAL CONST Robtarget Tr_meulage_bavure_186 := [[-74.393171875,-170.861875,115.7181875],[0.664342210232796,-0.745754209264803,0.0373350594183178,-0.033259290507512],[0,0,0,0],[8.999999E+09,8.999999E+09,8.999999E+09,8.999999E+09,8.999999E+09,8.999999E+09]];
    LOCAL CONST Robtarget Tr_meulage_bavure_187 := [[-78.797,-171.009796875,115.6621171875],[0.664260014710169,-0.742413059617728,0.0648896184499899,-0.0580587563051784],[0,0,0,0],[8.999999E+09,8.999999E+09,8.999999E+09,8.999999E+09,8.999999E+09,8.999999E+09]];
    LOCAL CONST Robtarget Tr_meulage_bavure_188 := [[-82.182375,-171.167953125,115.62525],[0.662080783578478,-0.736251193928903,0.104054925890418,-0.0935723669269605],[0,0,0,0],[8.999999E+09,8.999999E+09,8.999999E+09,8.999999E+09,8.999999E+09,8.999999E+09]];
    LOCAL CONST Robtarget Tr_meulage_bavure_189 := [[-84.573234375,-171.137078125,115.5791796875],[0.655720077793463,-0.724982094298341,0.156331012883739,-0.141395745820271],[0,0,0,0],[8.999999E+09,8.999999E+09,8.999999E+09,8.999999E+09,8.999999E+09,8.999999E+09]];
    LOCAL CONST Robtarget Tr_meulage_bavure_190 := [[-85.7801796875,-170.915921875,115.5270234375],[0.642820701224894,-0.706140192806145,0.219550199171385,-0.199863163750204],[0,0,0,0],[8.999999E+09,8.999999E+09,8.999999E+09,8.999999E+09,8.999999E+09,8.999999E+09]];
    LOCAL CONST Robtarget Tr_meulage_bavure_191 := [[-88.4296953125,-170.001953125,115.3523125],[0.622677298774636,-0.679165656884641,0.286432430846953,-0.262608938648863],[0,0,0,0],[8.999999E+09,8.999999E+09,8.999999E+09,8.999999E+09,8.999999E+09,8.999999E+09]];
    LOCAL CONST Robtarget Tr_meulage_bavure_192 := [[-88.918734375,-169.7575,115.3094140625],[0.59780966906714,-0.647035231181266,0.347602075166483,-0.321156981116708],[0,0,0,0],[8.999999E+09,8.999999E+09,8.999999E+09,8.999999E+09,8.999999E+09,8.999999E+09]];
    LOCAL CONST Robtarget Tr_meulage_bavure_193 := [[-89.5302890625,-169.128015625,115.2102578125],[0.572599070440967,-0.614657773834966,0.396959103292613,-0.369796695371267],[0,0,0,0],[8.999999E+09,8.999999E+09,8.999999E+09,8.999999E+09,8.999999E+09,8.999999E+09]];
    LOCAL CONST Robtarget Tr_meulage_bavure_194 := [[-90.82709375,-167.168546875,114.9121953125],[0.550562080167402,-0.585917167506537,0.43333625111741,-0.407188116440509],[0,0,0,0],[8.999999E+09,8.999999E+09,8.999999E+09,8.999999E+09,8.999999E+09,8.999999E+09]];
    LOCAL CONST Robtarget Tr_meulage_bavure_195 := [[-91.2550625,-164.63821875,114.5490546875],[0.533328296037147,-0.562529509887272,0.458463241213938,-0.43466416416322],[0,0,0,0],[8.999999E+09,8.999999E+09,8.999999E+09,8.999999E+09,8.999999E+09,8.999999E+09]];
    LOCAL CONST Robtarget Tr_meulage_bavure_196 := [[-91.4672578125,-163.633859375,114.404171875],[0.52113633290675,-0.544698115558835,0.474762660368314,-0.454226046975688],[0,0,0,0],[8.999999E+09,8.999999E+09,8.999999E+09,8.999999E+09,8.999999E+09,8.999999E+09]];
    LOCAL CONST Robtarget Tr_meulage_bavure_197 := [[-91.51909375,-162.5861875,114.2560078125],[0.513476782883588,-0.531812863874034,0.48447013186794,-0.467766354695888],[0,0,0,0],[8.999999E+09,8.999999E+09,8.999999E+09,8.999999E+09,8.999999E+09,8.999999E+09]];
    LOCAL CONST Robtarget Tr_meulage_bavure_198 := [[-91.52096875,-159.049,113.75878125],[0.509441382419957,-0.522901238420717,0.489499996241142,-0.476899912367413],[0,0,0,0],[8.999999E+09,8.999999E+09,8.999999E+09,8.999999E+09,8.999999E+09,8.999999E+09]];
    LOCAL CONST Robtarget Tr_meulage_bavure_199 := [[-91.7426015625,-149.08965625,112.355],[0.508000342748599,-0.516854966712831,0.491426673707781,-0.483007680601552],[0,0,0,0],[8.999999E+09,8.999999E+09,8.999999E+09,8.999999E+09,8.999999E+09,8.999999E+09]];
    LOCAL CONST Robtarget Tr_meulage_bavure_200 := [[-91.8348125,-144.7829375,111.74803125],[0.508140378003591,-0.512619158725735,0.49153759557173,-0.487243005582686],[0,0,0,0],[8.999999E+09,8.999999E+09,8.999999E+09,8.999999E+09,8.999999E+09,8.999999E+09]];
    LOCAL CONST Robtarget Tr_meulage_bavure_201 := [[-91.8389765625,-144.529140625,111.7122890625],[0.509112906918896,-0.509495462321344,0.490703515923074,-0.490335070480672],[0,0,0,0],[8.999999E+09,8.999999E+09,8.999999E+09,8.999999E+09,8.999999E+09,8.999999E+09]];
    LOCAL CONST Robtarget Tr_meulage_bavure_202 := [[-91.88765625,-142.804734375,111.469046875],[0.510467181344449,-0.507001901556814,0.489431637162252,-0.492776826903119],[0,0,0,0],[8.999999E+09,8.999999E+09,8.999999E+09,8.999999E+09,8.999999E+09,8.999999E+09]];
    LOCAL CONST Robtarget Tr_meulage_bavure_203 := [[-92.20571875,-134.132203125,110.24446875],[0.511950565146148,-0.504920608024539,0.487998144167169,-0.494792491584167],[0,0,0,0],[8.999999E+09,8.999999E+09,8.999999E+09,8.999999E+09,8.999999E+09,8.999999E+09]];
    LOCAL CONST Robtarget Tr_meulage_bavure_204 := [[-92.437140625,-128.091046875,109.391265625],[0.513513875038866,-0.503217483653162,0.486462998510584,-0.49641657442962],[0,0,0,0],[8.999999E+09,8.999999E+09,8.999999E+09,8.999999E+09,8.999999E+09,8.999999E+09]];
    LOCAL CONST Robtarget Tr_meulage_bavure_205 := [[-92.4062109375,-124.699390625,108.9150703125],[0.515133800545837,-0.501864598956793,0.48485743128374,-0.497676966694333],[0,0,0,0],[8.999999E+09,8.999999E+09,8.999999E+09,8.999999E+09,8.999999E+09,8.999999E+09]];
    LOCAL CONST Robtarget Tr_meulage_bavure_206 := [[-92.4177109375,-124.066234375,108.825875],[0.516765681041449,-0.500824692429697,0.483231872923377,-0.498612891270806],[0,0,0,0],[8.999999E+09,8.999999E+09,8.999999E+09,8.999999E+09,8.999999E+09,8.999999E+09]];
    LOCAL CONST Robtarget Tr_meulage_bavure_207 := [[-92.4446640625,-122.960921875,108.6700390625],[0.51835274695851,-0.500013646053416,0.481647007218388,-0.499312471222687],[0,0,0,0],[8.999999E+09,8.999999E+09,8.999999E+09,8.999999E+09,8.999999E+09,8.999999E+09]];
    LOCAL CONST Robtarget Tr_meulage_bavure_208 := [[-92.8264296875,-112.1201484375,107.1395703125],[0.519811283004719,-0.499340820439732,0.480188574912774,-0.499873891723504],[0,0,0,0],[8.999999E+09,8.999999E+09,8.999999E+09,8.999999E+09,8.999999E+09,8.999999E+09]];
    LOCAL CONST Robtarget Tr_meulage_bavure_209 := [[-92.830203125,-112.0312265625,107.127],[0.521066998119485,-0.498741183898411,0.47893167417103,-0.50037072899011],[0,0,0,0],[8.999999E+09,8.999999E+09,8.999999E+09,8.999999E+09,8.999999E+09,8.999999E+09]];
    LOCAL CONST Robtarget Tr_meulage_bavure_210 := [[-93.0031484375,-107.6880546875,106.5135],[0.522116197142305,-0.498154658585711,0.477880125951919,-0.500866447300265],[0,0,0,0],[8.999999E+09,8.999999E+09,8.999999E+09,8.999999E+09,8.999999E+09,8.999999E+09]];
    LOCAL CONST Robtarget Tr_meulage_bavure_211 := [[-93.076734375,-105.0583046875,106.1425703125],[0.52296898208403,-0.497587096138133,0.477023912287433,-0.501356871540428],[0,0,0,0],[8.999999E+09,8.999999E+09,8.999999E+09,8.999999E+09,8.999999E+09,8.999999E+09]];
    LOCAL CONST Robtarget Tr_meulage_bavure_212 := [[-93.1549921875,-103.9338046875,105.983140625],[0.523673676458628,-0.49705517649447,0.476314958503253,-0.501822769920217],[0,0,0,0],[8.999999E+09,8.999999E+09,8.999999E+09,8.999999E+09,8.999999E+09,8.999999E+09]];
    LOCAL CONST Robtarget Tr_meulage_bavure_213 := [[-93.22978125,-101.9080390625,105.69709375],[0.524265277239487,-0.49659388765163,0.475718856433328,-0.502227039755736],[0,0,0,0],[8.999999E+09,8.999999E+09,8.999999E+09,8.999999E+09,8.999999E+09,8.999999E+09]];
    LOCAL CONST Robtarget Tr_meulage_bavure_214 := [[-93.5059375,-93.938109375,104.572],[0.524784706060274,-0.496210907086518,0.475195146030603,-0.502558773839002],[0,0,0,0],[8.999999E+09,8.999999E+09,8.999999E+09,8.999999E+09,8.999999E+09,8.999999E+09]];
    LOCAL CONST Robtarget Tr_meulage_bavure_215 := [[-93.582109375,-91.0201953125,104.1605234375],[0.525269345781913,-0.495896287369727,0.47470665316085,-0.502824601625245],[0,0,0,0],[8.999999E+09,8.999999E+09,8.999999E+09,8.999999E+09,8.999999E+09,8.999999E+09]];
    LOCAL CONST Robtarget Tr_meulage_bavure_216 := [[-93.6075,-90.6105234375,104.1024921875],[0.525704960499218,-0.495646707422378,0.474267786132131,-0.503029524943813],[0,0,0,0],[8.999999E+09,8.999999E+09,8.999999E+09,8.999999E+09,8.999999E+09,8.999999E+09]];
    LOCAL CONST Robtarget Tr_meulage_bavure_217 := [[-93.7213125,-86.71553125,103.553015625],[0.526064668205574,-0.49543062901343,0.473905086548836,-0.503208133523552],[0,0,0,0],[8.999999E+09,8.999999E+09,8.999999E+09,8.999999E+09,8.999999E+09,8.999999E+09]];
    LOCAL CONST Robtarget Tr_meulage_bavure_218 := [[-93.9356328125,-79.1293984375,102.482953125],[0.526315852831235,-0.495182044674137,0.473650130943107,-0.503430153197491],[0,0,0,0],[8.999999E+09,8.999999E+09,8.999999E+09,8.999999E+09,8.999999E+09,8.999999E+09]];
    LOCAL CONST Robtarget Tr_meulage_bavure_219 := [[-94.1089453125,-74.38846875,101.81353125],[0.526395659122284,-0.494840467999266,0.473564534359526,-0.503762992968251],[0,0,0,0],[8.999999E+09,8.999999E+09,8.999999E+09,8.999999E+09,8.999999E+09,8.999999E+09]];
    LOCAL CONST Robtarget Tr_meulage_bavure_220 := [[-94.1434921875,-71.753015625,101.442484375],[0.526263612153634,-0.494341112099808,0.473687037782477,-0.504275783324755],[0,0,0,0],[8.999999E+09,8.999999E+09,8.999999E+09,8.999999E+09,8.999999E+09,8.999999E+09]];
    LOCAL CONST Robtarget Tr_meulage_bavure_221 := [[-94.2286640625,-69.408921875,101.1115078125],[0.52590068479982,-0.493677482675896,0.474035478003611,-0.504976611755197],[0,0,0,0],[8.999999E+09,8.999999E+09,8.999999E+09,8.999999E+09,8.999999E+09,8.999999E+09]];
    LOCAL CONST Robtarget Tr_meulage_bavure_222 := [[-94.3160390625,-66.8883046875,100.7556796875],[0.525374376186989,-0.492886729486796,0.474541979511505,-0.505820468568884],[0,0,0,0],[8.999999E+09,8.999999E+09,8.999999E+09,8.999999E+09,8.999999E+09,8.999999E+09]];
    LOCAL CONST Robtarget Tr_meulage_bavure_223 := [[-94.4334375,-63.49651171875,100.2768671875],[0.524808570676422,-0.492084764195851,0.475084938725615,-0.506678250951197],[0,0,0,0],[8.999999E+09,8.999999E+09,8.999999E+09,8.999999E+09,8.999999E+09,8.999999E+09]];
    LOCAL CONST Robtarget Tr_meulage_bavure_224 := [[-94.58928125,-58.42791796875,99.5616953125],[0.524364544968693,-0.491433164502918,0.475508413176606,-0.507372661664668],[0,0,0,0],[8.999999E+09,8.999999E+09,8.999999E+09,8.999999E+09,8.999999E+09,8.999999E+09]];
    LOCAL CONST Robtarget Tr_meulage_bavure_225 := [[-94.67365625,-57.5092734375,99.43109375],[0.524210832647951,-0.491067658949732,0.475649964598988,-0.507752566163041],[0,0,0,0],[8.999999E+09,8.999999E+09,8.999999E+09,8.999999E+09,8.999999E+09,8.999999E+09]];
    LOCAL CONST Robtarget Tr_meulage_bavure_226 := [[-94.6802734375,-55.91699609375,99.2071640625],[0.524445047614033,-0.491054768954736,0.475415701347854,-0.507742569450163],[0,0,0,0],[8.999999E+09,8.999999E+09,8.999999E+09,8.999999E+09,8.999999E+09,8.999999E+09]];
    LOCAL CONST Robtarget Tr_meulage_bavure_227 := [[-94.8214921875,-50.89054296875,98.498171875],[0.525028019418793,-0.491389816088351,0.474844605499898,-0.507350202618942],[0,0,0,0],[8.999999E+09,8.999999E+09,8.999999E+09,8.999999E+09,8.999999E+09,8.999999E+09]];
    LOCAL CONST Robtarget Tr_meulage_bavure_228 := [[-94.917484375,-45.1065625,97.6834921875],[0.525838995981719,-0.491940974719576,0.474051830089511,-0.506717169716673],[0,0,0,0],[8.999999E+09,8.999999E+09,8.999999E+09,8.999999E+09,8.999999E+09,8.999999E+09]];
    LOCAL CONST Robtarget Tr_meulage_bavure_229 := [[-94.9421953125,-44.0853359375,97.5395078125],[0.526686282522187,-0.492526961514034,0.473222374077563,-0.506042820971809],[0,0,0,0],[8.999999E+09,8.999999E+09,8.999999E+09,8.999999E+09,8.999999E+09,8.999999E+09]];
    LOCAL CONST Robtarget Tr_meulage_bavure_230 := [[-94.9206796875,-42.117578125,97.263296875],[0.52738656614898,-0.492972025895341,0.472534673853074,-0.505522475797863],[0,0,0,0],[8.999999E+09,8.999999E+09,8.999999E+09,8.999999E+09,8.999999E+09,8.999999E+09]];
    LOCAL CONST Robtarget Tr_meulage_bavure_231 := [[-95.036234375,-39.8536953125,96.9430625],[0.527806544286431,-0.493149622955176,0.472119653461197,-0.505298658224284],[0,0,0,0],[8.999999E+09,8.999999E+09,8.999999E+09,8.999999E+09,8.999999E+09,8.999999E+09]];
    LOCAL CONST Robtarget Tr_meulage_bavure_232 := [[-95.1740390625,-34.03544921875,96.122828125],[0.527905623422383,-0.49301433309693,0.472017389852598,-0.50542269814162],[0,0,0,0],[8.999999E+09,8.999999E+09,8.999999E+09,8.999999E+09,8.999999E+09,8.999999E+09]];
    LOCAL CONST Robtarget Tr_meulage_bavure_233 := [[-95.347515625,-28.34328125,95.3196953125],[0.527718942604453,-0.492594375472888,0.472193027036317,-0.505862870832791],[0,0,0,0],[8.999999E+09,8.999999E+09,8.999999E+09,8.999999E+09,8.999999E+09,8.999999E+09]];
    LOCAL CONST Robtarget Tr_meulage_bavure_234 := [[-95.45796875,-24.9697265625,94.843578125],[0.527318755046925,-0.491962756800867,0.472575025105913,-0.506537680871619],[0,0,0,0],[8.999999E+09,8.999999E+09,8.999999E+09,8.999999E+09,8.999999E+09,8.999999E+09]];
    LOCAL CONST Robtarget Tr_meulage_bavure_235 := [[-95.509921875,-23.002064453125,94.56609375],[0.526793757459659,-0.491194703081902,0.473075552442158,-0.507361431769664],[0,0,0,0],[8.999999E+09,8.999999E+09,8.999999E+09,8.999999E+09,8.999999E+09,8.999999E+09]];
    LOCAL CONST Robtarget Tr_meulage_bavure_236 := [[-95.510984375,-20.497291015625,94.2139921875],[0.526222424904499,-0.490345208629495,0.473616910199977,-0.50827016268354],[0,0,0,0],[8.999999E+09,8.999999E+09,8.999999E+09,8.999999E+09,8.999999E+09,8.999999E+09]];
    LOCAL CONST Robtarget Tr_meulage_bavure_237 := [[-95.5551328125,-17.20926171875,93.7510546875],[0.525670312712743,-0.48946747583732,0.474134909196731,-0.509203692357918],[0,0,0,0],[8.999999E+09,8.999999E+09,8.999999E+09,8.999999E+09,8.999999E+09,8.999999E+09]];
    LOCAL CONST Robtarget Tr_meulage_bavure_238 := [[-95.9686953125,-9.769044921875,92.698015625],[0.525207280286278,-0.488611482327546,0.474561702929705,-0.510105206976393],[0,0,0,0],[8.999999E+09,8.999999E+09,8.999999E+09,8.999999E+09,8.999999E+09,8.999999E+09]];
    LOCAL CONST Robtarget Tr_meulage_bavure_239 := [[-96.03675,-7.9697119140625,92.4439140625],[0.524904531779684,-0.487842772089084,0.474829552975673,-0.510902689226149],[0,0,0,0],[8.999999E+09,8.999999E+09,8.999999E+09,8.999999E+09,8.999999E+09,8.999999E+09]];
    LOCAL CONST Robtarget Tr_meulage_bavure_240 := [[-96.0907265625,-6.65112744140625,92.257625],[0.524841353674886,-0.48720975232666,0.47486260915148,-0.511540529323295],[0,0,0,0],[8.999999E+09,8.999999E+09,8.999999E+09,8.999999E+09,8.999999E+09,8.999999E+09]];
    LOCAL CONST Robtarget Tr_meulage_bavure_241 := [[-96.0646796875,-2.67666723632813,91.699421875],[0.525054035954144,-0.48671462178265,0.474625907067729,-0.512013070742702],[0,0,0,0],[8.999999E+09,8.999999E+09,8.999999E+09,8.999999E+09,8.999999E+09,8.999999E+09]];
    LOCAL CONST Robtarget Tr_meulage_bavure_242 := [[-96.065125,-1.13720056152344,91.4830234375],[0.525499002500919,-0.486301740401438,0.474160912539555,-0.512379590413912],[0,0,0,0],[8.999999E+09,8.999999E+09,8.999999E+09,8.999999E+09,8.999999E+09,8.999999E+09]];
    LOCAL CONST Robtarget Tr_meulage_bavure_243 := [[-96.116078125,1.04091772460938,91.1759765625],[0.526063308274471,-0.48584850957463,0.473574162321518,-0.512772985065421],[0,0,0,0],[8.999999E+09,8.999999E+09,8.999999E+09,8.999999E+09,8.999999E+09,8.999999E+09]];
    LOCAL CONST Robtarget Tr_meulage_bavure_244 := [[-96.159984375,1.04094799804687,91.175203125],[0.526596383934702,-0.485192895753828,0.473006558772309,-0.513370137128455],[0,0,0,0],[8.999999E+09,8.999999E+09,8.999999E+09,8.999999E+09,8.999999E+09,8.999999E+09]];
    LOCAL CONST Robtarget Tr_meulage_bavure_245 := [[-96.167859375,3.899724609375,90.7732265625],[0.526967927138443,-0.484195343398847,0.472578088766206,-0.514324433812322],[0,0,0,0],[8.999999E+09,8.999999E+09,8.999999E+09,8.999999E+09,8.999999E+09,8.999999E+09]];
    LOCAL CONST Robtarget Tr_meulage_bavure_246 := [[-96.1972109375,8.4426337890625,90.13415625],[0.527118293839987,-0.482776342009974,0.472338846115626,-0.515722136760531],[0,0,0,0],[8.999999E+09,8.999999E+09,8.999999E+09,8.999999E+09,8.999999E+09,8.999999E+09]];
    LOCAL CONST Robtarget Tr_meulage_bavure_247 := [[-96.3110703125,13.123560546875,89.474203125],[0.527105156410618,-0.480982424418388,0.472227464906878,-0.517510659671442],[0,0,0,0],[8.999999E+09,8.999999E+09,8.999999E+09,8.999999E+09,8.999999E+09,8.999999E+09]];
    LOCAL CONST Robtarget Tr_meulage_bavure_248 := [[-96.364,15.766712890625,89.1017578125],[0.527097853925665,-0.478958871271288,0.472078943372735,-0.519526441330539],[0,0,0,0],[8.999999E+09,8.999999E+09,8.999999E+09,8.999999E+09,8.999999E+09,8.999999E+09]];
    LOCAL CONST Robtarget Tr_meulage_bavure_249 := [[-96.4462734375,19.5217109375,88.5725078125],[0.5272459394789,-0.476841805265618,0.471751140907866,-0.521617171023123],[0,0,0,0],[8.999999E+09,8.999999E+09,8.999999E+09,8.999999E+09,8.999999E+09,8.999999E+09]];
    LOCAL CONST Robtarget Tr_meulage_bavure_250 := [[-96.4369609375,19.782423828125,88.5360234375],[0.527581045356717,-0.4746669803517,0.471213994271898,-0.523743133555406],[0,0,0,0],[8.999999E+09,8.999999E+09,8.999999E+09,8.999999E+09,8.999999E+09,8.999999E+09]];
    LOCAL CONST Robtarget Tr_meulage_bavure_251 := [[-96.46515625,20.317994140625,88.46025],[0.527825496938867,-0.472188482344787,0.470715927890138,-0.52617943436882],[0,0,0,0],[8.999999E+09,8.999999E+09,8.999999E+09,8.999999E+09,8.999999E+09,8.999999E+09]];
    LOCAL CONST Robtarget Tr_meulage_bavure_252 := [[-96.484625,22.542017578125,88.147296875],[0.527204088810346,-0.468753549392007,0.470939247829521,-0.529662329723205],[0,0,0,0],[8.999999E+09,8.999999E+09,8.999999E+09,8.999999E+09,8.999999E+09,8.999999E+09]];
    LOCAL CONST Robtarget Tr_meulage_bavure_253 := [[-96.64415625,30.228984375,87.064015625],[0.524511504825345,-0.46334350813632,0.472894574974268,-0.535323449639269],[0,0,0,0],[8.999999E+09,8.999999E+09,8.999999E+09,8.999999E+09,8.999999E+09,8.999999E+09]];
    LOCAL CONST Robtarget Tr_meulage_bavure_254 := [[-96.7007734375,31.08171875,86.9431640625],[0.518153071906971,-0.454644946138234,0.477798129876704,-0.5445404614082],[0,0,0,0],[8.999999E+09,8.999999E+09,8.999999E+09,8.999999E+09,8.999999E+09,8.999999E+09]];
    LOCAL CONST Robtarget Tr_meulage_bavure_255 := [[-96.7346015625,32.688818359375,86.7166796875],[0.506325761162958,-0.441209359423602,0.486760147336035,-0.558599215632432],[0,0,0,0],[8.999999E+09,8.999999E+09,8.999999E+09,8.999999E+09,8.999999E+09,8.999999E+09]];
    LOCAL CONST Robtarget Tr_meulage_bavure_256 := [[-97.0675703125,37.7479296875,85.9997421875],[0.487181918495299,-0.421586563582406,0.500458181734096,-0.578325302951048],[0,0,0,0],[8.999999E+09,8.999999E+09,8.999999E+09,8.999999E+09,8.999999E+09,8.999999E+09]];
    LOCAL CONST Robtarget Tr_meulage_bavure_257 := [[-96.80259375,40.82314453125,85.572109375],[0.459031591901888,-0.394528304028934,0.518851426348146,-0.603680886174613],[0,0,0,0],[8.999999E+09,8.999999E+09,8.999999E+09,8.999999E+09,8.999999E+09,8.999999E+09]];
    LOCAL CONST Robtarget Tr_meulage_bavure_258 := [[-96.566546875,41.527828125,85.4771796875],[0.420863395321502,-0.359367964277506,0.540855197455919,-0.633406918271672],[0,0,0,0],[8.999999E+09,8.999999E+09,8.999999E+09,8.999999E+09,8.999999E+09,8.999999E+09]];
    LOCAL CONST Robtarget Tr_meulage_bavure_259 := [[-95.822390625,44.22005859375,85.1117421875],[0.373133153765245,-0.316665923616772,0.564275815208132,-0.664896342862808],[0,0,0,0],[8.999999E+09,8.999999E+09,8.999999E+09,8.999999E+09,8.999999E+09,8.999999E+09]];
    LOCAL CONST Robtarget Tr_meulage_bavure_260 := [[-95.64853125,44.90273828125,85.0188203125],[0.318747079512612,-0.269017731424137,0.586193867990702,-0.694554899638387],[0,0,0,0],[8.999999E+09,8.999999E+09,8.999999E+09,8.999999E+09,8.999999E+09,8.999999E+09]];
    LOCAL CONST Robtarget Tr_meulage_bavure_261 := [[-95.6023125,45.025375,85.002390625],[0.263072212738095,-0.220962987624302,0.60401376230639,-0.719121508459944],[0,0,0,0],[8.999999E+09,8.999999E+09,8.999999E+09,8.999999E+09,8.999999E+09,8.999999E+09]];
    LOCAL CONST Robtarget Tr_meulage_bavure_262 := [[-91.31040625,48.50034765625,84.5888515625],[0.212217188804125,-0.177543404864132,0.616615863333459,-0.737039402780379],[0,0,0,0],[8.999999E+09,8.999999E+09,8.999999E+09,8.999999E+09,8.999999E+09,8.999999E+09]];
    LOCAL CONST Robtarget Tr_meulage_bavure_263 := [[-91.2993984375,48.51134765625,84.5875],[0.170679719568103,-0.142367929027074,0.624520504004076,-0.748714863076185],[0,0,0,0],[8.999999E+09,8.999999E+09,8.999999E+09,8.999999E+09,8.999999E+09,8.999999E+09]];
    LOCAL CONST Robtarget Tr_meulage_bavure_264 := [[-91.2787265625,48.5176328125,84.5869765625],[0.140260420186884,-0.116764615377166,0.629054169569785,-0.75563476023254],[0,0,0,0],[8.999999E+09,8.999999E+09,8.999999E+09,8.999999E+09,8.999999E+09,8.999999E+09]];
    LOCAL CONST Robtarget Tr_meulage_bavure_265 := [[-87.8363828125,49.27466015625,84.54065625],[0.12064465011355,-0.100348053981805,0.631550202701218,-0.759288797447384],[0,0,0,0],[8.999999E+09,8.999999E+09,8.999999E+09,8.999999E+09,8.999999E+09,8.999999E+09]];
    LOCAL CONST Robtarget Tr_meulage_bavure_266 := [[-87.8234765625,49.27529296875,84.5407890625],[0.110535622381351,-0.0919617202615354,0.632917160254841,-0.760750147187797],[0,0,0,0],[8.999999E+09,8.999999E+09,8.999999E+09,8.999999E+09,8.999999E+09,8.999999E+09]];
    LOCAL CONST Robtarget Tr_meulage_bavure_267 := [[-87.73859375,49.29593359375,84.5393671875],[0.108752458213319,-0.0905974604465095,0.633616774349427,-0.760588447359169],[0,0,0,0],[8.999999E+09,8.999999E+09,8.999999E+09,8.999999E+09,8.999999E+09,8.999999E+09]];
    LOCAL CONST Robtarget Tr_meulage_bavure_268 := [[-84.773828125,49.95,84.4991796875],[0.11503959522081,-0.0960623842473675,0.633716599425598,-0.758907887346415],[0,0,0,0],[8.999999E+09,8.999999E+09,8.999999E+09,8.999999E+09,8.999999E+09,8.999999E+09]];
    LOCAL CONST Robtarget Tr_meulage_bavure_269 := [[-82.883515625,50.2249453125,84.49353125],[0.13015020447378,-0.109039327489473,0.632876452854653,-0.755406344134194],[0,0,0,0],[8.999999E+09,8.999999E+09,8.999999E+09,8.999999E+09,8.999999E+09,8.999999E+09]];
    LOCAL CONST Robtarget Tr_meulage_bavure_270 := [[-76.189125,51.8800078125,84.3777421875],[0.155361862804346,-0.130695641383829,0.630338685130904,-0.749302664439861],[0,0,0,0],[8.999999E+09,8.999999E+09,8.999999E+09,8.999999E+09,8.999999E+09,8.999999E+09]];
    LOCAL CONST Robtarget Tr_meulage_bavure_271 := [[-75.845625,52.2978359375,84.3250078125],[0.191449362780329,-0.161824046787733,0.624931306146678,-0.739338205404032],[0,0,0,0],[8.999999E+09,8.999999E+09,8.999999E+09,8.999999E+09,8.999999E+09,8.999999E+09]];
    LOCAL CONST Robtarget Tr_meulage_bavure_272 := [[-75.596390625,52.74933203125,84.2658984375],[0.23730052727412,-0.201641018853083,0.61533226185865,-0.724151618645732],[0,0,0,0],[8.999999E+09,8.999999E+09,8.999999E+09,8.999999E+09,8.999999E+09,8.999999E+09]];
    LOCAL CONST Robtarget Tr_meulage_bavure_273 := [[-74.63259375,54.19496484375,84.079515625],[0.289131701051216,-0.247060061222159,0.600814151120423,-0.703126262779011],[0,0,0,0],[8.999999E+09,8.999999E+09,8.999999E+09,8.999999E+09,8.999999E+09,8.999999E+09]];
    LOCAL CONST Robtarget Tr_meulage_bavure_274 := [[-74.377828125,55.12261328125,83.9535703125],[0.341362767175181,-0.293356537387517,0.582012325398233,-0.677255532456584],[0,0,0,0],[8.999999E+09,8.999999E+09,8.999999E+09,8.999999E+09,8.999999E+09,8.999999E+09]];
    LOCAL CONST Robtarget Tr_meulage_bavure_275 := [[-73.1758671875,57.33415625,83.6636953125],[0.388989763342398,-0.336164126983744,0.560830401242163,-0.648960634234957],[0,0,0,0],[8.999999E+09,8.999999E+09,8.999999E+09,8.999999E+09,8.999999E+09,8.999999E+09]];
    LOCAL CONST Robtarget Tr_meulage_bavure_276 := [[-72.9423671875,58.77347265625,83.465453125],[0.429318086130583,-0.372994873347621,0.539460879988958,-0.620920900227319],[0,0,0,0],[8.999999E+09,8.999999E+09,8.999999E+09,8.999999E+09,8.999999E+09,8.999999E+09]];
    LOCAL CONST Robtarget Tr_meulage_bavure_277 := [[-72.8190546875,60.84019921875,83.1771015625],[0.461712018857951,-0.403089586200146,0.519655369694424,-0.59523028643279],[0,0,0,0],[8.999999E+09,8.999999E+09,8.999999E+09,8.999999E+09,8.999999E+09,8.999999E+09]];
    LOCAL CONST Robtarget Tr_meulage_bavure_278 := [[-72.6282890625,63.8663671875,82.7550703125],[0.486623273232709,-0.426637300543251,0.50257284929879,-0.573235496878157],[0,0,0,0],[8.999999E+09,8.999999E+09,8.999999E+09,8.999999E+09,8.999999E+09,8.999999E+09]];
    LOCAL CONST Robtarget Tr_meulage_bavure_279 := [[-72.8562109375,74.5178828125,81.253890625],[0.504826977044926,-0.444124764428805,0.488923535840243,-0.555748767853077],[0,0,0,0],[8.999999E+09,8.999999E+09,8.999999E+09,8.999999E+09,8.999999E+09,8.999999E+09]];
    LOCAL CONST Robtarget Tr_meulage_bavure_280 := [[-72.88871875,75.5807734375,81.103921875],[0.517106810308566,-0.456088986672306,0.479092830034906,-0.543188220765027],[0,0,0,0],[8.999999E+09,8.999999E+09,8.999999E+09,8.999999E+09,8.999999E+09,8.999999E+09]];
    LOCAL CONST Robtarget Tr_meulage_bavure_281 := [[-72.9544765625,77.4453203125,80.8406875],[0.524139588075091,-0.463011951376316,0.473215822598436,-0.535690591981654],[0,0,0,0],[8.999999E+09,8.999999E+09,8.999999E+09,8.999999E+09,8.999999E+09,8.999999E+09]];
    LOCAL CONST Robtarget Tr_meulage_bavure_282 := [[-72.96559375,77.9778671875,80.7656328125],[0.526418246456824,-0.465262887115032,0.471270316430774,-0.533215307846601],[0,0,0,0],[8.999999E+09,8.999999E+09,8.999999E+09,8.999999E+09,8.999999E+09,8.999999E+09]];
    !
    !Declaration des points de tronconnage

    !Tronconnage_0 : Tronconnage0
    LOCAL CONST Robtarget Tronconnage_0 := [[97.617015625,-37.65166796875,83.8049765625],[0.0010893607855984,0.0113405026984008,-0.707015836455272,-0.707105942057539],[0,0,0,0],[8.999999E+09,8.999999E+09,8.999999E+09,8.999999E+09,8.999999E+09,8.999999E+09]];

    !Tronconnage_1 : Tronconnage1
    LOCAL CONST Robtarget Tronconnage_1 := [[-54.14878125,-136.973,5.124578125],[0.174044837583629,0.605636307715718,-0.364972139726408,-0.685352751880729],[0,0,0,0],[8.999999E+09,8.999999E+09,8.999999E+09,8.999999E+09,8.999999E+09,8.999999E+09]];

    !
    !Cycle
    LOCAL PROC Cycle()
        !
        Prise;
        !
        Tronconnage;
        !
        Meulage;
        !
        !
        Depose;
        !
    ENDPROC

    !Trajectoire de prise de la pièce
    LOCAL PROC PRISE()

		!
        !Trigger localisation
        LocalisationPieceTable 700 \model:=0;
        !
        !Approche
		MoveJ Reltool(PicKPosition,0,0,-200),V1000,Z0,Tool_Prehenseur \Wobj:=Wobj_vision;
		MoveL Reltool(PicKPosition,0,0,-100),V500,Z0,Tool_Prehenseur \Wobj:=Wobj_vision;
		MoveL Reltool(PicKPosition,0,0,-10),V200,Z0,Tool_Prehenseur \Wobj:=Wobj_vision;
		MoveL PicKPosition,V100,Fine,Tool_Prehenseur \Wobj:=Wobj_vision;

        !Fermeture pince
		Gripper_Close;
        !
		MoveL Reltool(PicKPosition,0,0,-200),V500,Z0,Tool_Prehenseur \Wobj:=Wobj_vision;

        !Trigger relocalisation
		LocalisationPiecePrehenseur 700 \model:=0,Ref;
        !
        PEO;
        !
    ENDPROC

    !Trajectoire de tronconnage
    LOCAL PROC Tronconnage()
        !
        !StartMotor1();
        !
        ConfJ \Off;
        ConfL \Off;

        !Trajectoire
            !---------- tronconnage zone : 1 ------------

            !Approche PLAN

            MoveAbsJ [[0,-40,40,0,90,0],[9E9,9E9,9E9,9E9,9E9,9E9]]\NoEOffs,V500,Z0,Tool_Prehenseur;
            Tool := ToolOffset(Tool_M2_D490_S180);
            !
            !Approche
            MoveJ Reltool(Tronconnage_0,-200,0,-300),V1000,Z0,Tool \Wobj:=Wobj_Part_0;
            MoveL Reltool(Tronconnage_0,0,0,-300),V500,Z0,Tool \Wobj:=Wobj_Part_0;
            MoveL Reltool(Tronconnage_0,0,0,-200),V500,Z0,Tool \Wobj:=Wobj_Part_0;
            MoveL Reltool(Tronconnage_0,0,0,-150),V100,Z0,Tool \Wobj:=Wobj_Part_0;
            !
            Movel reltool(Tronconnage_0,0,0,-36.0493828125),V100,Z0,Tool \Wobj:=Wobj_Part_0;
            Movel Tronconnage_0,V100,Z0,Tool \Wobj:=Wobj_Part_0;
            Movel reltool(Tronconnage_0,0,0,36.0493828125),V100,Z0,Tool \Wobj:=Wobj_Part_0;
            !
            !Degagement
            MoveL Reltool(Tronconnage_0,0,0,-150),V100,Z0,Tool \Wobj:=Wobj_Part_0;
            MoveL Reltool(Tronconnage_0,0,0,-200),V500,Z0,Tool \Wobj:=Wobj_Part_0;
            MoveL Reltool(Tronconnage_0,0,0,-300),V500,Z0,Tool \Wobj:=Wobj_Part_0;
            MoveJ Reltool(Tronconnage_0,-200,0,-300),V1000,Z0,Tool \Wobj:=Wobj_Part_0;

            !Degagement PLAN

            MoveAbsJ [[0,-40,40,0,90,0],[9E9,9E9,9E9,9E9,9E9,9E9]]\NoEOffs,V500,Z0,Tool_Prehenseur;
            !
            !
        !Trajectoire
            !---------- tronconnage zone : 1 ------------

            !Approche DESSUS

            !Appel approche dessus;
            MoveAbsJ [[0,-40,40,0,90,0],[9E9,9E9,9E9,9E9,9E9,9E9]]\NoEOffs,V500,Z0,Tool_Prehenseur;
            Tool := ToolOffset(Tool_M2_D490_S180);
            !
            !Approche
            MoveJ Reltool(Tronconnage_1,-200,0,-300),V1000,Z0,Tool \Wobj:=Wobj_Part_0;
            MoveL Reltool(Tronconnage_1,0,0,-300),V500,Z0,Tool \Wobj:=Wobj_Part_0;
            MoveL Reltool(Tronconnage_1,0,0,-200),V500,Z0,Tool \Wobj:=Wobj_Part_0;
            MoveL Reltool(Tronconnage_1,0,0,-150),V100,Z0,Tool \Wobj:=Wobj_Part_0;
            !
            Movel reltool(Tronconnage_1,0,0,-23.19321875),V100,Z0,Tool \Wobj:=Wobj_Part_0;
            Movel Tronconnage_1,V100,Z0,Tool \Wobj:=Wobj_Part_0;
            Movel reltool(Tronconnage_1,0,0,23.19321875),V100,Z0,Tool \Wobj:=Wobj_Part_0;
            !
            !Degagement
            MoveL Reltool(Tronconnage_1,0,0,-150),V100,Z0,Tool \Wobj:=Wobj_Part_0;
            MoveL Reltool(Tronconnage_1,0,0,-200),V500,Z0,Tool \Wobj:=Wobj_Part_0;
            MoveL Reltool(Tronconnage_1,0,0,-300),V500,Z0,Tool \Wobj:=Wobj_Part_0;
            MoveJ Reltool(Tronconnage_1,-200,0,-300),V1000,Z0,Tool \Wobj:=Wobj_Part_0;

            !Degagement DESSUS

            !Appel approche dessus;
            MoveAbsJ [[0,-40,40,0,90,0],[9E9,9E9,9E9,9E9,9E9,9E9]]\NoEOffs,V500,Z0,Tool_Prehenseur;
            !
            !

    ENDPROC


    !Trajectoire de meulage
    LOCAL PROC Meulage()
        !
        !StartMotor2();
        !

        ConfJ \Off;
        ConfL \Off;


        !---------- Meulage zone : 1 ------------

        !Approche PLAN

        MoveAbsJ [[0,-40,40,0,90,0],[9E9,9E9,9E9,9E9,9E9,9E9]]\NoEOffs,V500,Z0,Tool_Prehenseur;

        !
        !Approche
        MoveJ Reltool(Tr_meulage_motif_1_0,0,0,-200),V1000,Z0,Tool_M1_D500_S0 \Wobj:=Wobj_Part_0;
        MoveL Reltool(Tr_meulage_motif_1_0,0,0,-100),V500,Z0,Tool_M1_D500_S0 \Wobj:=Wobj_Part_0;
        MoveL Reltool(Tr_meulage_motif_1_0,0,0,-10),V100,Z0,Tool_M1_D500_S0 \Wobj:=Wobj_Part_0;
        !
        !Trajectoire
        Movel Tr_meulage_motif_1_0,VitesseLente,Z0,Tool_M1_D500_S0 \Wobj:=Wobj_Part_0;
        Movel Tr_meulage_motif_1_1,VitesseLente,Z0,Tool_M1_D500_S0 \Wobj:=Wobj_Part_0;
        Movel Tr_meulage_motif_1_2,VitesseLente,Z0,Tool_M1_D500_S0 \Wobj:=Wobj_Part_0;
        Movel Tr_meulage_motif_1_3,VitesseLente,Z0,Tool_M1_D500_S0 \Wobj:=Wobj_Part_0;
        Movel Tr_meulage_motif_1_4,VitesseLente,Z0,Tool_M1_D500_S0 \Wobj:=Wobj_Part_0;
        Movel Tr_meulage_motif_1_5,VitesseLente,Z0,Tool_M1_D500_S0 \Wobj:=Wobj_Part_0;
        Movel Tr_meulage_motif_1_6,VitesseLente,Z0,Tool_M1_D500_S0 \Wobj:=Wobj_Part_0;
        Movel Tr_meulage_motif_1_7,VitesseLente,Z0,Tool_M1_D500_S0 \Wobj:=Wobj_Part_0;
        Movel Tr_meulage_motif_1_8,VitesseLente,Z0,Tool_M1_D500_S0 \Wobj:=Wobj_Part_0;
        Movel Tr_meulage_motif_1_9,VitesseLente,Z0,Tool_M1_D500_S0 \Wobj:=Wobj_Part_0;
        Movel Tr_meulage_motif_1_10,VitesseLente,Z0,Tool_M1_D500_S0 \Wobj:=Wobj_Part_0;
        Movel Tr_meulage_motif_1_11,VitesseLente,Z0,Tool_M1_D500_S0 \Wobj:=Wobj_Part_0;
        Movel Tr_meulage_motif_1_12,VitesseLente,Z0,Tool_M1_D500_S0 \Wobj:=Wobj_Part_0;
        Movel Tr_meulage_motif_1_13,VitesseLente,Z0,Tool_M1_D500_S0 \Wobj:=Wobj_Part_0;
        Movel Tr_meulage_motif_1_14,VitesseLente,Z0,Tool_M1_D500_S0 \Wobj:=Wobj_Part_0;
        Movel Tr_meulage_motif_1_15,VitesseLente,Z0,Tool_M1_D500_S0 \Wobj:=Wobj_Part_0;
        Movel Tr_meulage_motif_1_16,VitesseLente,Z0,Tool_M1_D500_S0 \Wobj:=Wobj_Part_0;
        Movel Tr_meulage_motif_1_17,VitesseLente,Z0,Tool_M1_D500_S0 \Wobj:=Wobj_Part_0;
        Movel Tr_meulage_motif_1_18,VitesseLente,Z0,Tool_M1_D500_S0 \Wobj:=Wobj_Part_0;
        Movel Tr_meulage_motif_1_19,VitesseLente,Z0,Tool_M1_D500_S0 \Wobj:=Wobj_Part_0;
        Movel Tr_meulage_motif_1_20,VitesseLente,Z0,Tool_M1_D500_S0 \Wobj:=Wobj_Part_0;
        Movel Tr_meulage_motif_1_21,VitesseLente,Z0,Tool_M1_D500_S0 \Wobj:=Wobj_Part_0;
        Movel Tr_meulage_motif_1_22,VitesseLente,Z0,Tool_M1_D500_S0 \Wobj:=Wobj_Part_0;
        Movel Tr_meulage_motif_1_23,VitesseLente,Z0,Tool_M1_D500_S0 \Wobj:=Wobj_Part_0;
        Movel Tr_meulage_motif_1_24,VitesseLente,Z0,Tool_M1_D500_S0 \Wobj:=Wobj_Part_0;
        Movel Tr_meulage_motif_1_25,VitesseLente,Z0,Tool_M1_D500_S0 \Wobj:=Wobj_Part_0;
        Movel Tr_meulage_motif_1_26,VitesseLente,Z0,Tool_M1_D500_S0 \Wobj:=Wobj_Part_0;
        Movel Tr_meulage_motif_1_27,VitesseLente,Z0,Tool_M1_D500_S0 \Wobj:=Wobj_Part_0;
        Movel Tr_meulage_motif_1_28,VitesseLente,Z0,Tool_M1_D500_S0 \Wobj:=Wobj_Part_0;
        Movel Tr_meulage_motif_1_29,VitesseLente,Z0,Tool_M1_D500_S0 \Wobj:=Wobj_Part_0;
        Movel Tr_meulage_motif_1_30,VitesseLente,Z0,Tool_M1_D500_S0 \Wobj:=Wobj_Part_0;
        Movel Tr_meulage_motif_1_31,VitesseLente,Z0,Tool_M1_D500_S0 \Wobj:=Wobj_Part_0;
        Movel Tr_meulage_motif_1_32,VitesseLente,Z0,Tool_M1_D500_S0 \Wobj:=Wobj_Part_0;
        Movel Tr_meulage_motif_1_33,VitesseLente,Z0,Tool_M1_D500_S0 \Wobj:=Wobj_Part_0;
        Movel Tr_meulage_motif_1_34,VitesseLente,Z0,Tool_M1_D500_S0 \Wobj:=Wobj_Part_0;
        Movel Tr_meulage_motif_1_35,VitesseLente,Z0,Tool_M1_D500_S0 \Wobj:=Wobj_Part_0;
        Movel Tr_meulage_motif_1_36,VitesseLente,Z0,Tool_M1_D500_S0 \Wobj:=Wobj_Part_0;
        Movel Tr_meulage_motif_1_37,VitesseLente,Z0,Tool_M1_D500_S0 \Wobj:=Wobj_Part_0;
        Movel Tr_meulage_motif_1_38,VitesseLente,Z0,Tool_M1_D500_S0 \Wobj:=Wobj_Part_0;
        Movel Tr_meulage_motif_1_39,VitesseLente,Z0,Tool_M1_D500_S0 \Wobj:=Wobj_Part_0;
        Movel Tr_meulage_motif_1_40,VitesseLente,Z0,Tool_M1_D500_S0 \Wobj:=Wobj_Part_0;
        Movel Tr_meulage_motif_1_41,VitesseLente,Z0,Tool_M1_D500_S0 \Wobj:=Wobj_Part_0;
        Movel Tr_meulage_motif_1_42,VitesseLente,Z0,Tool_M1_D500_S0 \Wobj:=Wobj_Part_0;
        Movel Tr_meulage_motif_1_43,VitesseLente,Z0,Tool_M1_D500_S0 \Wobj:=Wobj_Part_0;
        Movel Tr_meulage_motif_1_44,VitesseLente,Z0,Tool_M1_D500_S0 \Wobj:=Wobj_Part_0;
        Movel Tr_meulage_motif_1_45,VitesseLente,Z0,Tool_M1_D500_S0 \Wobj:=Wobj_Part_0;
        Movel Tr_meulage_motif_1_46,VitesseLente,Z0,Tool_M1_D500_S0 \Wobj:=Wobj_Part_0;
        Movel Tr_meulage_motif_1_47,VitesseLente,Z0,Tool_M1_D500_S0 \Wobj:=Wobj_Part_0;
        Movel Tr_meulage_motif_1_48,VitesseLente,Z0,Tool_M1_D500_S0 \Wobj:=Wobj_Part_0;
        Movel Tr_meulage_motif_1_49,VitesseLente,Z0,Tool_M1_D500_S0 \Wobj:=Wobj_Part_0;
        Movel Tr_meulage_motif_1_50,VitesseLente,Z0,Tool_M1_D500_S0 \Wobj:=Wobj_Part_0;
        Movel Tr_meulage_motif_1_51,VitesseLente,Z0,Tool_M1_D500_S0 \Wobj:=Wobj_Part_0;
        Movel Tr_meulage_motif_1_52,VitesseLente,Z0,Tool_M1_D500_S0 \Wobj:=Wobj_Part_0;
        Movel Tr_meulage_motif_1_53,VitesseLente,Z0,Tool_M1_D500_S0 \Wobj:=Wobj_Part_0;
        Movel Tr_meulage_motif_1_54,VitesseLente,Z0,Tool_M1_D500_S0 \Wobj:=Wobj_Part_0;
        Movel Tr_meulage_motif_1_55,VitesseLente,Z0,Tool_M1_D500_S0 \Wobj:=Wobj_Part_0;
        Movel Tr_meulage_motif_1_56,VitesseLente,Z0,Tool_M1_D500_S0 \Wobj:=Wobj_Part_0;
        Movel Tr_meulage_motif_1_57,VitesseLente,Z0,Tool_M1_D500_S0 \Wobj:=Wobj_Part_0;
        Movel Tr_meulage_motif_1_58,VitesseLente,Z0,Tool_M1_D500_S0 \Wobj:=Wobj_Part_0;
        Movel Tr_meulage_motif_1_59,VitesseLente,Z0,Tool_M1_D500_S0 \Wobj:=Wobj_Part_0;
        Movel Tr_meulage_motif_1_60,VitesseLente,Z0,Tool_M1_D500_S0 \Wobj:=Wobj_Part_0;
        Movel Tr_meulage_motif_1_61,VitesseLente,Z0,Tool_M1_D500_S0 \Wobj:=Wobj_Part_0;
        Movel Tr_meulage_motif_1_62,VitesseLente,Z0,Tool_M1_D500_S0 \Wobj:=Wobj_Part_0;
        Movel Tr_meulage_motif_1_63,VitesseLente,Z0,Tool_M1_D500_S0 \Wobj:=Wobj_Part_0;
        Movel Tr_meulage_motif_1_64,VitesseLente,Z0,Tool_M1_D500_S0 \Wobj:=Wobj_Part_0;
        Movel Tr_meulage_motif_1_65,VitesseLente,Z0,Tool_M1_D500_S0 \Wobj:=Wobj_Part_0;
        Movel Tr_meulage_motif_1_66,VitesseLente,Z0,Tool_M1_D500_S0 \Wobj:=Wobj_Part_0;
        Movel Tr_meulage_motif_1_67,VitesseLente,Z0,Tool_M1_D500_S0 \Wobj:=Wobj_Part_0;
        Movel Tr_meulage_motif_1_68,VitesseLente,Z0,Tool_M1_D500_S0 \Wobj:=Wobj_Part_0;
        Movel Tr_meulage_motif_1_69,VitesseLente,Z0,Tool_M1_D500_S0 \Wobj:=Wobj_Part_0;
        Movel Tr_meulage_motif_1_70,VitesseLente,Z0,Tool_M1_D500_S0 \Wobj:=Wobj_Part_0;
        Movel Tr_meulage_motif_1_71,VitesseLente,Z0,Tool_M1_D500_S0 \Wobj:=Wobj_Part_0;
        Movel Tr_meulage_motif_1_72,VitesseLente,Z0,Tool_M1_D500_S0 \Wobj:=Wobj_Part_0;
        Movel Tr_meulage_motif_1_73,VitesseLente,Z0,Tool_M1_D500_S0 \Wobj:=Wobj_Part_0;
        Movel Tr_meulage_motif_1_74,VitesseLente,Z0,Tool_M1_D500_S0 \Wobj:=Wobj_Part_0;
        Movel Tr_meulage_motif_1_75,VitesseLente,Z0,Tool_M1_D500_S0 \Wobj:=Wobj_Part_0;
        Movel Tr_meulage_motif_1_76,VitesseLente,Z0,Tool_M1_D500_S0 \Wobj:=Wobj_Part_0;
        Movel Tr_meulage_motif_1_77,VitesseLente,Z0,Tool_M1_D500_S0 \Wobj:=Wobj_Part_0;
        Movel Tr_meulage_motif_1_78,VitesseLente,Z0,Tool_M1_D500_S0 \Wobj:=Wobj_Part_0;
        Movel Tr_meulage_motif_1_79,VitesseLente,Z0,Tool_M1_D500_S0 \Wobj:=Wobj_Part_0;
        Movel Tr_meulage_motif_1_80,VitesseLente,Z0,Tool_M1_D500_S0 \Wobj:=Wobj_Part_0;
        Movel Tr_meulage_motif_1_81,VitesseLente,Z0,Tool_M1_D500_S0 \Wobj:=Wobj_Part_0;
        Movel Tr_meulage_motif_1_82,VitesseLente,Z0,Tool_M1_D500_S0 \Wobj:=Wobj_Part_0;
        Movel Tr_meulage_motif_1_83,VitesseLente,Z0,Tool_M1_D500_S0 \Wobj:=Wobj_Part_0;
        Movel Tr_meulage_motif_1_84,VitesseLente,Z0,Tool_M1_D500_S0 \Wobj:=Wobj_Part_0;
        Movel Tr_meulage_motif_1_85,VitesseLente,Z0,Tool_M1_D500_S0 \Wobj:=Wobj_Part_0;
        Movel Tr_meulage_motif_1_86,VitesseLente,Z0,Tool_M1_D500_S0 \Wobj:=Wobj_Part_0;
        Movel Tr_meulage_motif_1_87,VitesseLente,Z0,Tool_M1_D500_S0 \Wobj:=Wobj_Part_0;
        Movel Tr_meulage_motif_1_88,VitesseLente,Z0,Tool_M1_D500_S0 \Wobj:=Wobj_Part_0;
        Movel Tr_meulage_motif_1_89,VitesseLente,Z0,Tool_M1_D500_S0 \Wobj:=Wobj_Part_0;
        Movel Tr_meulage_motif_1_90,VitesseLente,Z0,Tool_M1_D500_S0 \Wobj:=Wobj_Part_0;
        Movel Tr_meulage_motif_1_91,VitesseLente,Z0,Tool_M1_D500_S0 \Wobj:=Wobj_Part_0;
        Movel Tr_meulage_motif_1_92,VitesseLente,Z0,Tool_M1_D500_S0 \Wobj:=Wobj_Part_0;
        Movel Tr_meulage_motif_1_93,VitesseLente,Z0,Tool_M1_D500_S0 \Wobj:=Wobj_Part_0;
        Movel Tr_meulage_motif_1_94,VitesseLente,Z0,Tool_M1_D500_S0 \Wobj:=Wobj_Part_0;
        Movel Tr_meulage_motif_1_95,VitesseLente,Z0,Tool_M1_D500_S0 \Wobj:=Wobj_Part_0;
        Movel Tr_meulage_motif_1_96,VitesseLente,Z0,Tool_M1_D500_S0 \Wobj:=Wobj_Part_0;
        Movel Tr_meulage_motif_1_97,VitesseLente,Z0,Tool_M1_D500_S0 \Wobj:=Wobj_Part_0;
        Movel Tr_meulage_motif_1_98,VitesseLente,Z0,Tool_M1_D500_S0 \Wobj:=Wobj_Part_0;
        Movel Tr_meulage_motif_1_99,VitesseLente,Z0,Tool_M1_D500_S0 \Wobj:=Wobj_Part_0;
        Movel Tr_meulage_motif_1_100,VitesseLente,Z0,Tool_M1_D500_S0 \Wobj:=Wobj_Part_0;
        Movel Tr_meulage_motif_1_101,VitesseLente,Z0,Tool_M1_D500_S0 \Wobj:=Wobj_Part_0;
        Movel Tr_meulage_motif_1_102,VitesseLente,Z0,Tool_M1_D500_S0 \Wobj:=Wobj_Part_0;
        Movel Tr_meulage_motif_1_103,VitesseLente,Z0,Tool_M1_D500_S0 \Wobj:=Wobj_Part_0;
        Movel Tr_meulage_motif_1_104,VitesseLente,Z0,Tool_M1_D500_S0 \Wobj:=Wobj_Part_0;
        Movel Tr_meulage_motif_1_105,VitesseLente,Z0,Tool_M1_D500_S0 \Wobj:=Wobj_Part_0;
        Movel Tr_meulage_motif_1_106,VitesseLente,Z0,Tool_M1_D500_S0 \Wobj:=Wobj_Part_0;
        Movel Tr_meulage_motif_1_107,VitesseLente,Z0,Tool_M1_D500_S0 \Wobj:=Wobj_Part_0;
        Movel Tr_meulage_motif_1_108,VitesseLente,Z0,Tool_M1_D500_S0 \Wobj:=Wobj_Part_0;
        Movel Tr_meulage_motif_1_109,VitesseLente,Z0,Tool_M1_D500_S0 \Wobj:=Wobj_Part_0;
        Movel Tr_meulage_motif_1_110,VitesseLente,Z0,Tool_M1_D500_S0 \Wobj:=Wobj_Part_0;
        Movel Tr_meulage_motif_1_111,VitesseLente,Z0,Tool_M1_D500_S0 \Wobj:=Wobj_Part_0;
        Movel Tr_meulage_motif_1_112,VitesseLente,Z0,Tool_M1_D500_S0 \Wobj:=Wobj_Part_0;
        Movel Tr_meulage_motif_1_113,VitesseLente,Z0,Tool_M1_D500_S0 \Wobj:=Wobj_Part_0;
        Movel Tr_meulage_motif_1_114,VitesseLente,Z0,Tool_M1_D500_S0 \Wobj:=Wobj_Part_0;
        Movel Tr_meulage_motif_1_115,VitesseLente,Z0,Tool_M1_D500_S0 \Wobj:=Wobj_Part_0;
        Movel Tr_meulage_motif_1_116,VitesseLente,Z0,Tool_M1_D500_S0 \Wobj:=Wobj_Part_0;
        Movel Tr_meulage_motif_1_117,VitesseLente,Z0,Tool_M1_D500_S0 \Wobj:=Wobj_Part_0;
        Movel Tr_meulage_motif_1_118,VitesseLente,Z0,Tool_M1_D500_S0 \Wobj:=Wobj_Part_0;
        Movel Tr_meulage_motif_1_119,VitesseLente,Z0,Tool_M1_D500_S0 \Wobj:=Wobj_Part_0;
        Movel Tr_meulage_motif_1_120,VitesseLente,Z0,Tool_M1_D500_S0 \Wobj:=Wobj_Part_0;
        !
        !Degagement
        MoveL Reltool(Tr_meulage_motif_1_120,0,0,-10),V100,Z0,Tool_M1_D500_S0 \Wobj:=Wobj_Part_0;
        MoveL Reltool(Tr_meulage_motif_1_120,0,0,-100),V500,Z0,Tool_M1_D500_S0 \Wobj:=Wobj_Part_0;
        MoveJ Reltool(Tr_meulage_motif_1_120,0,0,-200),V1000,Z0,Tool_M1_D500_S0 \Wobj:=Wobj_Part_0;


        MoveAbsJ [[0,-40,40,0,90,0],[9E9,9E9,9E9,9E9,9E9,9E9]]\NoEOffs,V500,Z0,Tool_Prehenseur;
        !
        !

        !---------- Meulage zone : 2 ------------

        !Approche DESSOUS

        MoveAbsJ [[0,-40,40,0,90,0],[9E9,9E9,9E9,9E9,9E9,9E9]]\NoEOffs,V500,Z0,Tool_Prehenseur;

